// TwinCAT 3 PLC project WF03
// ProgramVersion: 3.1.4024.0
// libraries:
//   Tc2_Standard, * (Beckhoff Automation GmbH)
//   Tc2_System, * (Beckhoff Automation GmbH)
//   Tc3_Module, * (Beckhoff Automation GmbH)
// project tree:
//   DUTs/ E_ServoStateMachine.TcDUT, E_State.TcTLEO, E_ComponentMode.TcTLEO (not stored), E_LenzeJogFreq.TcTLEO, E_RotationDirection.TcTLEO (not stored)
//   GVLs/ GVL.TcGVL
//   / PlcTask.TcTTO (not stored), RevolutionCounter.TcTTO
//   POUs/deprecated/ FB_Module_4posArm_Old.TcPOU (not stored), FB_Module_CoilHolder_Old.TcPOU, FB_Module_ToolHolderDoor_Old.TcPOU, FB_Module_ToolHolder_Old.TcPOU
//   POUs/FB_Components/ FB_Component_ACmotor.TcPOU, FB_Component_DualValve.TcPOU, FB_Component_DualValveGuarded.TcPOU, FB_Component_InductiveSensor.TcPOU, FB_Component_ReedSwitch.TcPOU, FB_Component_Servo.TcPOU, FB_Component_SingleValve.TcPOU, FB_Component_SingleValveGuarded.TcPOU, FB_Component_4posArm.TcPOU
//   POUs/ COUNTER.TcPOU, FB_Component_ServoMotor.TcPOU, FB_Module_CoilPusher.TcPOU, FB_Section_Cutter.TcPOU, FB_Section_ToolStation_Old.TcPOU, I_Component.TcIO, I_Module.TcIO, I_Section.TcIO, MAIN.TcPOU
//   POUs/FB_Modules/ FB_Module_CoilHolder.TcPOU, FB_Module_ToolHolder.TcPOU, FB_Module_ToolHolderDoor.TcPOU, FB_Module_Winder.TcPOU
// real-time tasks:
//   TASK PlcTask: cycle T#10ms, priority 20, ADS port 350
//   TASK RevolutionCounter: cycle T#2ms, priority 1, ADS port 351
// I/O:
//   DEVICE Device 1 (EtherCAT), AmsNetId 5.155.196.195.2.1
//     Term 1 (EK1200) [EK1200-5000 EtherCAT Power supply (2A E-Bus)]
//       Term 2 (EL1809) [EL1809 16Ch. Dig. Input 24V, 3ms]
//       Term 3 (EL1809) [EL1809 16Ch. Dig. Input 24V, 3ms]
//       Term 4 (EL1809) [EL1809 16Ch. Dig. Input 24V, 3ms]
//       Term 5 (EL1809) [EL1809 16Ch. Dig. Input 24V, 3ms]
//       Term 6 (EL2809) [EL2809 16Ch. Dig. Output 24V, 0.5A]
//       Term 7 (EL2809) [EL2809 16Ch. Dig. Output 24V, 0.5A]
//       Term 8 (EL2809) [EL2809 16Ch. Dig. Output 24V, 0.5A]
//       Term 20 (EL4032) [EL4032 2Ch. Ana. Output +/-10V, 12bit]
//       Term 21 (EL5112) [EL5112 2Ch. Inc. Encoder 5V (2xAB or 1xABC RS422,TTL)]
//       Term 21 (EL9011) [EL9011 End Terminal]
// variable links:
//   WF03/WF03 Instance <-> Device 1 (EtherCAT)/Term 1 (EK1200)/Term 2 (EL1809)
//     PlcTask Inputs/GVL.bDoorToolHolderDown <-> Channel 4/Input
//     PlcTask Inputs/GVL.bDoorToolHolderLock <-> Channel 3/Input
//     PlcTask Inputs/GVL.bWireClampRetracted <-> Channel 12/Input
//     PlcTask Inputs/GVL.bWireClampTransverse1Extended <-> Channel 14/Input
//     PlcTask Inputs/GVL.bWireClampTransverse2Extended <-> Channel 16/Input
//     PlcTask Inputs/GVL.bWireClampTransverse1Retracted <-> Channel 13/Input
//     PlcTask Inputs/GVL.bWireClampTransverse2Retracted <-> Channel 15/Input
//     PlcTask Inputs/GVL.bWirePusherDisengaged <-> Channel 1/Input
//     PlcTask Inputs/GVL.bWirePusherEngaged <-> Channel 2/Input
//   WF03/WF03 Instance <-> Device 1 (EtherCAT)/Term 1 (EK1200)/Term 20 (EL4032)
//     PlcTask Outputs/GVL.aOutServo1 <-> AO Outputs Channel 1/Analog output
//     PlcTask Outputs/GVL.aOutServo2 <-> AO Outputs Channel 2/Analog output
//   WF03/WF03 Instance <-> Device 1 (EtherCAT)/Term 1 (EK1200)/Term 21 (EL5112)
//     PlcTask Inputs/GVL.bSetCounterDoneServo1 <-> ENC Status Channel 2/Status/Set counter done
//     PlcTask Inputs/GVL.bSetCounterDoneServo2 <-> ENC Status Channel 1/Status/Set counter done
//     PlcTask Inputs/GVL.dCountServo1 <-> ENC Status Channel 2/Counter value
//     PlcTask Outputs/GVL.dSetCounterServo1 <-> ENC Control Channel 2/Control/Set counter
//     PlcTask Outputs/GVL.dSetCounterServo2 <-> ENC Control Channel 1/Control/Set counter
//     PlcTask Outputs/GVL.dSetCounterValueServo1 <-> ENC Control Channel 2/Set counter value
//     PlcTask Outputs/GVL.dSetCounterValueServo2 <-> ENC Control Channel 1/Set counter value
//     RevolutionCounter Inputs/GVL.dCountServo2 <-> ENC Status Channel 1/Counter value
//   WF03/WF03 Instance <-> Device 1 (EtherCAT)/Term 1 (EK1200)/Term 3 (EL1809)
//     PlcTask Inputs/GVL.bCoilHolderIndexBit{1..5} <-> Channel {1..5}/Input  (5 links)
//     PlcTask Inputs/GVL.bCoilHolderIndexReady <-> Channel 6/Input
//     PlcTask Inputs/GVL.bCoilHolderLocked <-> Channel 8/Input
//     PlcTask Inputs/GVL.bCoilHolderUnlocked <-> Channel 7/Input
//     PlcTask Inputs/GVL.bToolHolderIndexBit1 <-> Channel 9/Input
//     PlcTask Inputs/GVL.bToolHolderIndexBit2 <-> Channel 10/Input
//     PlcTask Inputs/GVL.bToolHolderLocked <-> Channel 12/Input
//     PlcTask Inputs/GVL.bToolHolderUnlocked <-> Channel 11/Input
//     PlcTask Inputs/GVL.bWireHolderPos{1..4} <-> Channel {13..16}/Input  (4 links)
//   WF03/WF03 Instance <-> Device 1 (EtherCAT)/Term 1 (EK1200)/Term 4 (EL1809)
//     PlcTask Inputs/GVL.bCoilPusherExtended <-> Channel 2/Input
//     PlcTask Inputs/GVL.bCoilPusherRetracted <-> Channel 1/Input
//     PlcTask Inputs/GVL.bMainPressureSense <-> Channel 16/Input
//     PlcTask Inputs/GVL.bWire{1..4}NotAvailable <-> Channel {5..8}/Input  (4 links)
//   WF03/WF03 Instance <-> Device 1 (EtherCAT)/Term 1 (EK1200)/Term 5 (EL1809)
//     PlcTask Inputs/GVL.bCoilTranslate <-> Channel 15/Input
//     PlcTask Inputs/GVL.bControlOnBtn <-> Channel 5/Input
//     PlcTask Inputs/GVL.bFeedBackSafetyRelay <-> Channel 6/Input
//     PlcTask Inputs/GVL.bLenze1Relay <-> Channel 13/Input
//     PlcTask Inputs/GVL.bLenze2Relay <-> Channel 14/Input
//     PlcTask Inputs/GVL.bReadyToOperate603 <-> Channel 11/Input
//     PlcTask Inputs/GVL.bReadyToOperate614 <-> Channel 12/Input
//     PlcTask Inputs/GVL.bSafetyContactBreakers <-> Channel 9/Input
//     PlcTask Inputs/GVL.bStartBtn <-> Channel 2/Input
//     PlcTask Inputs/GVL.bStartPosBtn <-> Channel 3/Input
//     PlcTask Inputs/GVL.bStopBtn <-> Channel 1/Input
//     PlcTask Inputs/GVL.bToolingRotationBtn <-> Channel 4/Input
//     RevolutionCounter Inputs/GVL.bCoilRotate <-> Channel 16/Input
//   WF03/WF03 Instance <-> Device 1 (EtherCAT)/Term 1 (EK1200)/Term 6 (EL2809)
//     PlcTask Outputs/GVL.b603Enable <-> Channel 9/Output
//     PlcTask Outputs/GVL.b614Enable <-> Channel 10/Output
//     PlcTask Outputs/GVL.bCloseToolCarrierDoor <-> Channel 15/Output
//     PlcTask Outputs/GVL.bLenze1Direction <-> Channel 4/Output
//     PlcTask Outputs/GVL.bLenze1InjectionBrake <-> Channel 3/Output
//     PlcTask Outputs/GVL.bLenze1JogBit1 <-> Channel 1/Output
//     PlcTask Outputs/GVL.bLenze1JogBit2 <-> Channel 2/Output
//     PlcTask Outputs/GVL.bLenze2JogBit1 <-> Channel 5/Output
//     PlcTask Outputs/GVL.bLenze2JogBit2 <-> Channel 6/Output
//     PlcTask Outputs/GVL.bLenze2njectionBrake <-> Channel 7/Output
//     PlcTask Outputs/GVL.bOpenToolCarrierDoor <-> Channel 14/Output
//     PlcTask Outputs/GVL.bPushCoil <-> Channel 16/Output
//     PlcTask Outputs/GVL.bResetServosErrors <-> Channel 8/Output
//     PlcTask Outputs/GVL.bStartBtnLight <-> Channel 11/Output
//     PlcTask Outputs/GVL.bStartPosBtnLight <-> Channel 12/Output
//     PlcTask Outputs/GVL.bToolingRotationBtnLight <-> Channel 13/Output
//   WF03/WF03 Instance <-> Device 1 (EtherCAT)/Term 1 (EK1200)/Term 7 (EL2809)
//     PlcTask Outputs/GVL.bEngageWireClamp <-> Channel 12/Output
//     PlcTask Outputs/GVL.bExtendWireClamp <-> Channel 7/Output
//     PlcTask Outputs/GVL.bExtendWireHolder <-> Channel 5/Output
//     PlcTask Outputs/GVL.bExtendWireHolderTransverse1 <-> Channel 16/Output
//     PlcTask Outputs/GVL.bExtendWireHolderTransverse2 <-> Channel 9/Output
//     PlcTask Outputs/GVL.bLockDoor <-> Channel 2/Output
//     PlcTask Outputs/GVL.bReleaseWireClamp <-> Channel 11/Output
//     PlcTask Outputs/GVL.bRetractWireClamp <-> Channel 6/Output
//     PlcTask Outputs/GVL.bRetractWireHolder <-> Channel 4/Output
//     PlcTask Outputs/GVL.bRetractWireHolderTransverse1 <-> Channel 15/Output
//     PlcTask Outputs/GVL.bRetractWireHolderTransverse2 <-> Channel 8/Output
//     PlcTask Outputs/GVL.bUnlockCoilHolder <-> Channel 13/Output
//     PlcTask Outputs/GVL.bUnlockToolHolder <-> Channel 14/Output
//     PlcTask Outputs/GVL.bWirePusherForward <-> Channel 10/Output
//   WF03/WF03 Instance <-> Device 1 (EtherCAT)/Term 1 (EK1200)/Term 8 (EL2809)
//     PlcTask Outputs/GVL.bCutWire <-> Channel 1/Output

CONFIGURATION WF03
    RESOURCE PLC ON TwinCAT3
        TASK RevolutionCounter(INTERVAL := T#2ms, PRIORITY := 1);
        PROGRAM COUNTER WITH RevolutionCounter : COUNTER;
    END_RESOURCE
END_CONFIGURATION

// ---- DUTs/E_ServoStateMachine.TcDUT
{attribute 'qualified_only'}
{attribute 'strict'}
TYPE E_ServoStateMachine :
(
	IDLE			:= 0,
	HOMING          := 1,
	HOMED           := 2,
	RAMPUP          := 3,
	HOLD            := 4,
	RAMPDOWN        := 5,
	FAULT			:= 6
);
END_TYPE

// ---- DUTs/E_State.TcTLEO
{attribute 'qualified_only'}
{attribute 'strict'}
TYPE E_State :
(
	DISABLED	:= 0,
	READY		:= 1,
	BUSY		:= 2,
	DONE 		:= 3,
	HALTED		:= 4,
	TIMEOUT 	:= 5
);
END_TYPE

// ---- DUTs/E_LenzeJogFreq.TcTLEO
{attribute 'qualified_only'}
{attribute 'strict'}
TYPE E_LenzeJogFreq :
(
	FOFF 	:= 0,
	F1		:= 1,
	F2		:= 2,
	F3		:= 3
);
END_TYPE

// ---- GVLs/GVL.TcGVL
{attribute 'qualified_only'}
VAR_GLOBAL
	uRevCount1		: INT;
	uRevCount2		: DINT;
	bResetRevCount	: BOOL;

/////////////////////////////////////////////////////////////////////////////////////////////
// 									DIGITAL INPUTS								   		   //
/////////////////////////////////////////////////////////////////////////////////////////////
	//--------------------------------
	// TERM 2 : EL1809 Digital In
	//--------------------------------
	bWirePusherDisengaged			AT %I*	: BOOL;	// S5.18	term 2.1
	bWirePusherEngaged				AT %I*	: BOOL;	// S5.17	term 2.2
	bDoorToolHolderLock				AT %I*	: BOOL;	//			term 2.3
	bDoorToolHolderDown				AT %I*	: BOOL;	// S5.20	term 2.4
	// term 2.5-11 --> unused
	bWireClampRetracted				AT %I*	: BOOL;	// S5.28	term 2.12
	bWireClampTransverse1Extended	AT %I*	: BOOL;	// S5.29	term 2.14
	bWireClampTransverse1Retracted	AT %I*	: BOOL;	// S5.30	term 2.13
	bWireClampTransverse2Extended	AT %I*	: BOOL;	// S5.31	term 2.16
	bWireClampTransverse2Retracted	AT %I*	: BOOL;	// S5.32	term 2.15
	//--------------------------------
	// TERM 3 : EL1809 Digital In
	//--------------------------------
	bCoilHolderIndexBit1			AT %I*	: BOOL;	// S5.1		term 3.1
	bCoilHolderIndexBit2			AT %I*	: BOOL;	// S5.2		term 3.2
	bCoilHolderIndexBit3			AT %I*	: BOOL;	// S5.3		term 3.3
	bCoilHolderIndexBit4			AT %I*	: BOOL;	// S5.4		term 3.4
	bCoilHolderIndexBit5			AT %I*	: BOOL;	// S5.5		term 3.5
	bCoilHolderIndexReady			AT %I*	: BOOL;	// S5.6		term 3.6
	bCoilHolderUnlocked				AT %I*	: BOOL; // S5.8		term 3.7	
	bCoilHolderLocked				AT %I*	: BOOL; // S5.7		term 3.8
	bToolHolderIndexBit1			AT %I*	: BOOL; // S5.9		term 3.9
	bToolHolderIndexBit2			AT %I*	: BOOL; // S5.10	term 3.10
	bToolHolderUnlocked				AT %I*	: BOOL; // S5.12	term 3.11
	bToolHolderLocked   			AT %I*	: BOOL; // S5.11	term 3.12
	bWireHolderPos1					AT %I*	: BOOL; // S5.13	term 3.13
	bWireHolderPos2					AT %I*	: BOOL; // S5.14	term 3.14
	bWireHolderPos3					AT %I*	: BOOL; // S5.15	term 3.15
	bWireHolderPos4					AT %I*	: BOOL; // S5.16	term 3.16
	//--------------------------------
	// TERM 4 : EL1809 Digital In
	//--------------------------------
	bCoilPusherRetracted			AT %I*	: BOOL;	// S4.17	term 4.1
	bCoilPusherExtended				AT %I*	: BOOL;	// S4.18	term 4.2
	// term 4.3-4 --> unused
	bWire1NotAvailable				AT %I*	: BOOL;	// S4.21	term 4.5
	bWire2NotAvailable				AT %I*	: BOOL;	// S4.22	term 4.6
	bWire3NotAvailable				AT %I*	: BOOL;	// S4.23	term 4.7
	bWire4NotAvailable				AT %I*	: BOOL;	// S4.24	term 4.8
	// term 4.9-15 --> unused
	bMainPressureSense				AT %I*	: BOOL;	// S4.32	term 4.16
	//--------------------------------
	// TERM 5 : EL1809 Digital In
	//--------------------------------
	bStopBtn						AT %I*	: BOOL;	//			term 5.1
	bStartBtn						AT %I*	: BOOL;	//			term 5.2
	bStartPosBtn					AT %I*	: BOOL;	//			term 5.3
	bToolingRotationBtn				AT %I*	: BOOL;	//			term 5.4
	bControlOnBtn					AT %I*	: BOOL;	//			term 5.5
	bFeedBackSafetyRelay			AT %I*	: BOOL; //			term 5.6
	// term 5.7 check why connected to GND											// TODO!!
	// term 5.8	check what contactor K1.1 does and if also checks other stuff		// TODO!!
	bSafetyContactBreakers			AT %I*	: BOOL;	//			term 5.9
	// term 5.10 --> unused
	bReadyToOperate603				AT %I*	: BOOL;	//			term 5.11			// rename
	bReadyToOperate614				AT %I*	: BOOL;	//			term 5.12			// rename
	bLenze1Relay					AT %I*	: BOOL;	//			term 5.13			// rename
	bLenze2Relay					AT %I*	: BOOL;	//			term 5.14			// rename
	bCoilTranslate					AT %I*	: BOOL;	//			term 5.15			// rename
	bCoilRotate						AT %I*	: BOOL;	//			term 5.16			// rename

/////////////////////////////////////////////////////////////////////////////////////////////
// 									DIGITAL OUTPUTS								   		   //
/////////////////////////////////////////////////////////////////////////////////////////////
	//--------------------------------
	// TERM 6 : EL2809 Digital Out
	//--------------------------------
	bLenze1JogBit1					AT %Q*	: BOOL;	//			term 6.1
	bLenze1JogBit2					AT %Q*	: BOOL;	//			term 6.2
	bLenze1InjectionBrake			AT %Q*	: BOOL; //			term 6.3
	bLenze1Direction				AT %Q*	: BOOL;	//			term 6.4
	bLenze2JogBit1					AT %Q*	: BOOL;	//			term 6.5
	bLenze2JogBit2					AT %Q*	: BOOL;	//			term 6.6
	bLenze2njectionBrake			AT %Q*	: BOOL; //			term 6.7
	bResetServosErrors				AT %Q*	: BOOL; //			term 6.8
	b603Enable						AT %Q*	: BOOL;	//			term 6.9
	b614Enable						AT %Q*	: BOOL;	//			term 6.10
	bStartBtnLight					AT %Q*	: BOOL; //			term 6.11
	bStartPosBtnLight				AT %Q*	: BOOL; //			term 6.12
	bToolingRotationBtnLight		AT %Q*	: BOOL; //			term 6.13
	bOpenToolCarrierDoor			AT %Q*	: BOOL; // Y6.4		term 6.14
	bCloseToolCarrierDoor			AT %Q*	: BOOL; // Y6.5		term 6.15
	bPushCoil						AT %Q*	: BOOL; // Y6.9		term 6.16
	//--------------------------------
	// TERM 7 : EL2809 Digital Out
	//--------------------------------
	// term 7.1 --> unused
	bLockDoor						AT %Q*	: BOOL; //			term 7.2
	// term 7.3 --> unused
	bRetractWireHolder				AT %Q*	: BOOL; // Y6.13	term 7.4
	bExtendWireHolder				AT %Q*	: BOOL; // Y6.14	term 7.5
	bRetractWireClamp				AT %Q*	: BOOL; // Y7.10	term 7.6		// pushes forward clamp
	bExtendWireClamp				AT %Q*	: BOOL; // Y7.11	term 7.7
	bRetractWireHolderTransverse2	AT %Q*	: BOOL; // Y7.7		term 7.8
	bExtendWireHolderTransverse2	AT %Q*	: BOOL; // Y7.8		term 7.9
	bWirePusherForward				AT %Q*	: BOOL; // Y7.9		term 7.10		// bent thingy pushing the wire at the top
	bReleaseWireClamp				AT %Q*	: BOOL; // Y6.15	term 7.11		// clamps wire
	bEngageWireClamp				AT %Q*	: BOOL; // Y6.16	term 7.12
	bUnlockCoilHolder				AT %Q*	: BOOL; // Y7.12	term 7.13
	bUnlockToolHolder				AT %Q*	: BOOL; // Y7.13	term 7.14
	bRetractWireHolderTransverse1	AT %Q*	: BOOL; // Y7.14	term 7.15
	bExtendWireHolderTransverse1	AT %Q*	: BOOL; // Y7.15	term 7.16
	//--------------------------------
	// TERM 8 : EL2809 Digital Out
	//--------------------------------
	bCutWire						AT %Q*	: BOOL; // Y8.1		term 7.1
	// term 8.2-9 --> unused
	// term 8.16-16 --> free
	
	//--------------------------------
	// TERM 8 : EL4032 Analog Out
	//--------------------------------
	aOutServo1						AT %Q*	: INT;	// term 20
	aOutServo2						AT %Q*	: INT;	// term 20
	
	bSetCounterDoneServo1			AT %I*	: BOOL;	// term 21
	dCountServo1					AT %I*	: DINT;	// term 21
	bSetCounterDoneServo2			AT %I*	: BOOL;	// term 21
	dCountServo2					AT %I*	: DINT;	// term 21
	
	dSetCounterServo1				AT %Q*	: BOOL;	// term 21
	dSetCounterValueServo1			AT %Q*	: DINT;	// term 21
	dSetCounterServo2				AT %Q*	: BOOL;	// term 21
	dSetCounterValueServo2			AT %Q*	: DINT;	// term 21
	
END_VAR

// ---- POUs/I_Component.TcIO
INTERFACE I_Component
VAR_INPUT
END_VAR

VAR_OUTPUT
END_VAR

METHOD M_Disable : BOOL
VAR_INPUT
END_VAR
END_METHOD

METHOD M_Enable : BOOL
VAR_INPUT
END_VAR
END_METHOD

METHOD M_Halt : BOOL
VAR_INPUT
END_VAR
END_METHOD

METHOD M_Resume : BOOL
VAR_INPUT
END_VAR
END_METHOD

END_INTERFACE

// ---- POUs/I_Module.TcIO
INTERFACE I_Module

METHOD M_Disable : BOOL
VAR_INPUT
END_VAR
END_METHOD

METHOD M_Enable : BOOL
VAR_INPUT
END_VAR
END_METHOD

METHOD M_Halt : BOOL
VAR_INPUT
END_VAR
END_METHOD

METHOD M_Resume : BOOL
VAR_INPUT
END_VAR
END_METHOD

END_INTERFACE

// ---- POUs/I_Section.TcIO
INTERFACE I_Section

METHOD M_Disable : BOOL
VAR_INPUT
END_VAR
END_METHOD

METHOD M_Enable : BOOL
VAR_INPUT
END_VAR
END_METHOD

METHOD M_Halt : BOOL
VAR_INPUT
END_VAR
END_METHOD

METHOD M_Resume : BOOL
VAR_INPUT
END_VAR
END_METHOD

END_INTERFACE

// ---- POUs/COUNTER.TcPOU
PROGRAM COUNTER
VAR
	tSensorTrig		: F_TRIG;
END_VAR

tSensorTrig(CLK := GVL.bCoilRotate);
IF tSensorTrig.Q THEN
	GVL.uRevCount1 := GVL.uRevCount1 + 1;
END_IF

IF GVL.bResetRevCount THEN
	GVL.bResetRevCount  := FALSE;
	GVL.uRevCount1		:= 0;
END_IF

GVL.uRevCount2 := REAL_TO_DINT(DINT_TO_REAL(GVL.dCountServo2) / 9216);

END_PROGRAM

// ---- POUs/deprecated/FB_Module_CoilHolder_Old.TcPOU
FUNCTION_BLOCK FB_Module_CoilHolder_Old IMPLEMENTS I_Module
VAR_INPUT
	bEnable			: BOOL;
END_VAR
VAR_OUTPUT
END_VAR
VAR
	Components		: ARRAY [0..9] OF I_Component;

	fbACmotor		: FB_Component_ACmotor;
	fbCoilLock		: FB_Component_SingleValve;
	fbReedLock		: FB_Component_ReedSwitch;
	fbReedUnlock	: FB_Component_ReedSwitch;
	
	fbIndexBit1		: FB_Component_InductiveSensor;
	fbIndexBit2		: FB_Component_InductiveSensor;
	fbIndexBit3		: FB_Component_InductiveSensor;
	fbIndexBit4		: FB_Component_InductiveSensor;
	fbIndexBit5		: FB_Component_InductiveSensor;
	fbIndexReady	: FB_Component_InductiveSensor;
	
	nIndex			: INT;
	idx				: INT;
END_VAR

IF bEnable THEN
	fbACmotor(
		bDeviceActive 	:= GVL.bLenze1Relay,
		sName			:= 'AC motor plate',
		bEnable			:= TRUE,
		bE1jog1			:= GVL.bLenze1JogBit1,
		bE2jog2			:= GVL.bLenze1JogBit2,
		bE3DCbrake		:= GVL.bLenze1InjectionBrake,
		eE4Direction	:= GVL.bLenze1Direction);
		
	fbCoilLock(
		sName 	:= 'Coil Lock',
		bEnable := TRUE,
		bOutput := GVL.bUnlockCoilHolder);
		
	fbReedLock(
		bRawSignal	:= GVL.bCoilHolderLocked,
		tDebounce	:= T#5MS,
		tTimeout	:= T#0S,
		sName		:= 'plate locked reed',
		bEnable		:= TRUE);
		
	fbReedUnlock(
		bRawSignal	:= GVL.bCoilHolderUnlocked,
		tDebounce	:= T#5MS,
		tTimeout	:= T#0S,
		sName		:= 'plate unlocked reed',
		bEnable		:= TRUE);
		
	fbIndexBit1(bRawSignal := GVL.bCoilHolderIndexBit1,
		tDebounce 	:= T#5MS,
		tTimeout	:= T#0S,
		sName		:= 'plate index 1',
		bEnable		:= TRUE);
		
	fbIndexBit2(bRawSignal := GVL.bCoilHolderIndexBit2,
		tDebounce 	:= T#5MS,
		tTimeout	:= T#0S,
		sName		:= 'plate index 2',
		bEnable		:= TRUE);
		
	fbIndexBit3(bRawSignal := GVL.bCoilHolderIndexBit3,
		tDebounce 	:= T#5MS,
		tTimeout	:= T#0S,
		sName		:= 'plate index 3',
		bEnable		:= TRUE);
		
	fbIndexBit4(bRawSignal := GVL.bCoilHolderIndexBit4,
		tDebounce 	:= T#5MS,
		tTimeout	:= T#0S,
		sName		:= 'plate index 4',
		bEnable		:= TRUE);
		
	fbIndexBit5(bRawSignal := GVL.bCoilHolderIndexBit5,
		tDebounce 	:= T#5MS,
		tTimeout	:= T#0S,
		sName		:= 'plate index 5',
		bEnable		:= TRUE);
		
	fbIndexReady(bRawSignal := GVL.bCoilHolderIndexReady,
		tDebounce 	:= T#5MS,
		tTimeout	:= T#0S,
		sName		:= 'plate index ready',
		bEnable		:= TRUE);

	Components[0] := fbACmotor;
	Components[1] := fbCoilLock;
	Components[2] := fbReedLock;
	Components[3] := fbReedUnlock;
	Components[4] := fbIndexBit1;
	Components[5] := fbIndexBit2;
	Components[6] := fbIndexBit3;
	Components[7] := fbIndexBit4;
	Components[8] := fbIndexBit5;
	Components[9] := fbIndexReady;
	
	FOR idx := 0 TO 9 DO
    	Components[idx].M_Start();
	END_FOR;
	
	// when index ready bit is triggered, convert index bits to integer
	IF fbIndexReady.bSensorActive THEN
		nIndex := 	TO_INT(SHL(TO_UINT(fbIndexBit5.bSensorActive), 4) OR
					SHL(TO_UINT(fbIndexBit4.bSensorActive), 3) OR
					SHL(TO_UINT(fbIndexBit3.bSensorActive), 2) OR
					SHL(TO_UINT(fbIndexBit2.bSensorActive), 1) OR
					(TO_UINT(fbIndexBit1.bSensorActive)));
	END_IF
END_IF

METHOD M_GoTo : BOOL
VAR_INPUT
	nTargetIndex	: INT;
END_VAR

VAR
	cwSteps: INT;
	target: INT;
	ccwSteps: INT;
	shortestDistance : INT;
END_VAR
IF fbReedUnlock.bSensorActive THEN
	IF nTargetIndex = nIndex THEN									// if target index is reached, turn off motor, lock plate and signal done
		fbACmotor.M_SetFreq(Frequency := E_LenzeJogFreq.F0FF);
		M_Lock();
		M_GoTo := TRUE;
		RETURN;
	END_IF
	
	cwSteps  := (nTargetIndex - nIndex + 24) MOD 24;				// calculate how much cw & ccw steps needed to go to target
	ccwSteps := (nIndex - nTargetIndex + 24) MOD 24;
	
	IF cwSteps <= ccwSteps THEN										// set direction for shortest path to target
		fbACmotor.M_SetDir(Direction := E_RotationDirection.CW);
		shortestDistance := cwSteps;
	ELSE
		fbACmotor.M_SetDir(Direction := E_RotationDirection.CCW);	
		shortestDistance := ccwSteps;
	END_IF
	
	IF nIndex <> nTargetIndex THEN
		IF shortestDistance <= 1 THEN								// if 1 from the target, set speed to slowest
			fbACmotor.M_SetFreq(Frequency := E_LenzeJogFreq.F1);	
		ELSIF shortestDistance <= 2 THEN							// if 2 from the target, set speed to slow
			fbACmotor.M_SetFreq(Frequency := E_LenzeJogFreq.F2);
		ELSE
			fbACmotor.M_SetFreq(Frequency := E_LenzeJogFreq.F3);	// if further set to highest speed
		END_IF
	ELSE
		fbACmotor.M_SetFreq(Frequency := E_LenzeJogFreq.F0FF);		// for safety, should be handled by first if
		M_Lock();
		M_GoTo := TRUE;
	END_IF
ELSE
	M_Unlock();														// unlock plate if locked
END_IF
END_METHOD

METHOD M_Halt : BOOL
VAR_INPUT
END_VAR
END_METHOD

METHOD M_Lock : BOOL
VAR_INPUT
END_VAR
fbCoilLock.M_Retract();
END_METHOD

METHOD M_Start : BOOL
VAR_INPUT
END_VAR
END_METHOD

METHOD M_Stop : BOOL
VAR_INPUT
END_VAR
END_METHOD

METHOD M_Unlock : BOOL
VAR_INPUT
END_VAR
fbCoilLock.M_Extend();
END_METHOD

END_FUNCTION_BLOCK

// ---- POUs/FB_Components/FB_Component_ACmotor.TcPOU
// Function block for AC motors controlled with the LENZE d-31855 frequency inverter
FUNCTION_BLOCK FB_Component_ACmotor IMPLEMENTS I_Component
VAR_INPUT
	sName			: STRING[50];
	tTimeout		: TIME := T#0MS;
END_VAR

VAR_OUTPUT
	eJogFreq		: E_LenzeJogFreq := E_LenzeJogFreq.FOFF;
	
	bEnabled     	: BOOL;
	eState			: E_State := E_State.DISABLED;
	eNextState		: E_State := E_State.DISABLED;
	sStatusText 	: STRING[100];
END_VAR

VAR_IN_OUT
	bDeviceActive	: BOOL;	
	bE1jog1			: BOOL;					// jog func b1
	bE2jog2			: BOOL;					// jog func b2
	bE3DCbrake		: BOOL;					// DC injection brake
	eE4Direction	: BOOL;					// motor direction
END_VAR

VAR
	bLastE1jog1		: BOOL;
	bLastE2jog2		: BOOL;
	eLastState		: E_State;
	tTimeoutTimer	: TON;
END_VAR


VAR CONSTANT
	DISABLED		: E_State := E_State.DISABLED;
	READY			: E_State := E_State.READY;
	BUSY			: E_State := E_State.BUSY;
	HALTED			: E_State := E_State.HALTED;
	TIMEOUT			: E_State := E_State.TIMEOUT;
	
	FOFF	: E_LenzeJogFreq := E_LenzeJogFreq.FOFF;
	F1		: E_LenzeJogFreq := E_LenzeJogFreq.F1;
	F2		: E_LenzeJogFreq := E_LenzeJogFreq.F2;
	F3		: E_LenzeJogFreq := E_LenzeJogFreq.F3;
END_VAR

tTimeoutTimer(PT := tTimeout);

eState := eNextState;

CASE eState OF
	DISABLED:	sStatusText := 'AC motor disabled';
	
	READY:	 	sStatusText := 'Motor not moving, waiting for instruction';
				IF NOT bDeviceActive THEN
					sStatusText := 'frequency inverter is not activated, please check if control is on and doors are closed';
				ELSIF eJogFreq <> FOFF THEN
					eNextState := BUSY;
				END_IF
				
	BUSY: 		M_ApplyFreq();
				CASE eJogFreq OF
					FOFF: 	eNextState	:= E_State.TIMEOUT;
					F1: 	sStatusText := CONCAT('motor running ', CONCAT(SEL(eE4Direction = TRUE, 'CCW','CW'), ' at freq 1'));		
					F2: 	sStatusText := CONCAT('motor running ', CONCAT(SEL(eE4Direction = TRUE, 'CCW','CW'), ' at freq 2'));				
					F3: 	sStatusText := CONCAT('motor running ', CONCAT(SEL(eE4Direction = TRUE, 'CCW','CW'), ' at freq 3')); 	
				END_CASE
	
	TIMEOUT: 	sStatusText := 'motor in timeout';
				tTimeoutTimer(IN := TRUE);
				
				IF tTimeoutTimer.Q THEN
					tTimeoutTimer(IN := FALSE);
					eNextState := READY;
				END_IF
	
	HALTED: 	sStatusText := 'motor halted';

END_CASE

METHOD M_ApplyFreq : BOOL
VAR_INPUT
END_VAR
IF eState = BUSY AND bDeviceActive THEN
	CASE eJogFreq OF
		FOFF: 	bE1jog1 	:= FALSE;
				bE2jog2 	:= FALSE;
				
		F1: 	bE1jog1 	:= TRUE;
				bE2jog2 	:= FALSE;
				
		F2: 	bE1jog1 	:= TRUE;
				bE2jog2 	:= TRUE;

		F3: 	bE1jog1 	:= FALSE;
				bE2jog2 	:= TRUE;
	END_CASE
END_IF
END_METHOD

METHOD M_Disable : BOOL
VAR_INPUT
END_VAR
IF eState = READY THEN
	bE1jog1		 	:= FALSE;
	bE2jog2		 	:= FALSE;
	bE3DCbrake 		:= FALSE;
	eE4Direction 	:= FALSE;
	tTimeoutTimer(IN := FALSE);	

	bEnabled	:= FALSE;
	eNextState	:= DISABLED;
END_IF
END_METHOD

METHOD M_Enable : BOOL
VAR_INPUT
END_VAR
IF eState = DISABLED THEN
	bEnabled	:= TRUE;
	eNextState 	:= READY;
END_IF
END_METHOD

METHOD M_Halt : BOOL
VAR_INPUT
END_VAR
IF eState <> HALTED AND eState <> DISABLED THEN
	bLastE1jog1 := bE1jog1;
	bLastE2jog2 := bE2jog2;
	
	bE1jog1		:= FALSE;
	bE2jog2		:= FALSE;
	bE3DCbrake	:= TRUE;
	
	eLastState 	:= eState;
	eNextState 	:= HALTED;	
END_IF
END_METHOD

METHOD M_Resume : BOOL
VAR_INPUT
END_VAR
IF eState = HALTED THEN
	bE1jog1 	:= bLastE1jog1;
	bE2jog2 	:= bLastE2jog2;
	bE3DCbrake 	:= FALSE;
	
	eNextState 	:= eLastState;
END_IF
END_METHOD

METHOD M_SetDir : BOOL
VAR_INPUT
	Direction: E_RotationDirection;
END_VAR
IF eState = READY THEN
	eE4Direction := TO_BOOL(Direction);
END_IF
END_METHOD

METHOD M_SetFreq : BOOL
VAR_INPUT
	Frequency: E_LenzeJogFreq;
END_VAR
IF eState = READY OR eState = BUSY THEN
	eJogFreq := Frequency;
END_IF
END_METHOD

END_FUNCTION_BLOCK

// ---- POUs/FB_Components/FB_Component_SingleValve.TcPOU
FUNCTION_BLOCK FB_Component_SingleValve IMPLEMENTS I_Component
VAR_INPUT
	sName			: STRING[50];
	tTimeout		: TIME := T#0S;
END_VAR

VAR_IN_OUT
	bOutput			: BOOL;
END_VAR

VAR_OUTPUT
	bEnabled     	: BOOL;
	eState			: E_State := E_State.DISABLED;
	eNextState		: E_State := E_State.DISABLED;
	sStatusText 	: STRING[100];
END_VAR

VAR
	tTimeoutTimer	: TON;
	eLastState		: E_State;
END_VAR

VAR CONSTANT
	DISABLED		: E_State := E_State.DISABLED;
	READY			: E_State := E_State.READY;
	BUSY			: E_State := E_State.BUSY;
	HALTED			: E_State := E_State.HALTED;
	TIMEOUT			: E_State := E_State.TIMEOUT;
END_VAR

tTimeoutTimer(PT := tTimeout);

eState := eNextState;

CASE eState OF
	DISABLED: 	sStatusText := 'piston is disabled';
	READY: 		sStatusText := 'piston ready to operate';
	BUSY: 		sStatusText := 'piston busy';
	TIMEOUT:	sStatusText := 'piston in timeout';
				tTimeoutTimer(IN := TRUE);
				
				IF tTimeoutTimer.Q THEN
					tTimeoutTimer(IN := FALSE);
					eNextState := READY;
				END_IF
				
	HALTED:		sStatusText := 'piston halted';
END_CASE

METHOD M_Disable : BOOL
VAR_INPUT
END_VAR
IF eState = READY THEN
	bEnabled	:= FALSE;
	eNextState	:= DISABLED;
END_IF
END_METHOD

METHOD M_Enable : BOOL
VAR_INPUT
END_VAR
IF eState = DISABLED THEN
	bEnabled	:= TRUE;
	eNextState	:= READY;
END_IF
END_METHOD

METHOD M_Extend : BOOL
VAR_INPUT
END_VAR
IF eState = READY OR eState = BUSY THEN
	bOutput := TRUE;
END_IF
END_METHOD

METHOD M_Halt : BOOL
VAR_INPUT
END_VAR
IF eState <> HALTED AND eState <> DISABLED THEN
	eLastState := eState;
	eNextState := HALTED;
END_IF
END_METHOD

METHOD M_Resume : BOOL
VAR_INPUT
END_VAR
IF eState = HALTED THEN
	eNextState := eLastState;
END_IF
END_METHOD

METHOD M_Retract : BOOL
VAR_INPUT
END_VAR
IF eState = READY OR eState = BUSY THEN
	bOutput	:= FALSE;
END_IF
END_METHOD

END_FUNCTION_BLOCK

// ---- POUs/FB_Components/FB_Component_ReedSwitch.TcPOU
// function block for reed switch with the option of debouncing + rising and falling edge detection.
FUNCTION_BLOCK FB_Component_ReedSwitch IMPLEMENTS I_Component
VAR_INPUT
	sName			: STRING[50];
	bRawSignal		: BOOL;				
	tDebounce		: TIME := T#0MS;
	tTimeout		: TIME := T#0MS;
END_VAR

VAR_OUTPUT
	bSensorActive	: BOOL;
	bTimeout		: BOOL;
	bRisingEdge		: BOOL;
	bFallingEdge	: BOOL;
	
	bEnabled		: BOOL;
	eState			: E_State := E_State.DISABLED;
	eNextState		: E_State := E_State.DISABLED;
	sStatusText 	: STRING[100];
END_VAR

VAR
	tDebounceTimer		: TON;
	tTimeoutTimer		: TON;
	
	bLastStableSignal	: BOOL := bRawSignal;
	bPendingSignal		: BOOL;
	
	eLastState			: E_State;
END_VAR

VAR CONSTANT
	DISABLED	: E_State := E_State.DISABLED;
	READY		: E_State := E_State.READY;
	BUSY		: E_State := E_State.BUSY;
	DONE		: E_State := E_State.DONE;
	HALTED		: E_State := E_State.HALTED;
	TIMEOUT		: E_State := E_State.TIMEOUT;
END_VAR

tDebounceTimer.PT 	:= tDebounce;
tTimeoutTimer.PT	:= tTimeout;

eState := eNextState;

CASE eState OF
	DISABLED:	sStatusText := 'Sensor disabled';
				
	READY:		sStatusText := 'Sensor idle, waiting for read';
				IF bRawSignal <> bLastStableSignal THEN
					bPendingSignal 	:= bRawSignal;
					eNextState 		:= BUSY;
				ELSE
					tTimeoutTimer(IN := FALSE);
					tDebounceTimer(IN := FALSE);
				END_IF
				
	BUSY:		sStatusText := 'Sensor is debouncing';
				tDebounceTimer(IN := TRUE);
				IF bRawSignal <> bPendingSignal THEN
					eNextState := READY;
				END_IF

				IF tDebounceTimer.Q THEN
					eNextState := TIMEOUT;
				END_IF
	TIMEOUT:	sStatusText := 'Sensor timeout';
				tTimeoutTimer(IN := TRUE);
				
				bRisingEdge  := NOT bLastStableSignal AND bPendingSignal;
				bFallingEdge := bLastStableSignal AND NOT bPendingSignal;
					
				bLastStableSignal := bPendingSignal;
				bSensorActive	  := bLastStableSignal;
				
				IF tTimeoutTimer.Q THEN
					tTimeoutTimer(IN 	:= FALSE);
					tDebounceTimer(IN 	:= FALSE);
					eNextState := READY;
				END_IF
				
	HALTED:		sStatusText := 'Sensor halted';
								
END_CASE

METHOD M_Disable : BOOL
VAR_INPUT
END_VAR
IF eState = READY THEN
	bEnabled	:= FALSE;
	eNextState	:= DISABLED;
END_IF
END_METHOD

METHOD M_Enable : BOOL
VAR_INPUT
END_VAR
IF eState = DISABLED THEN
	bEnabled	:= TRUE;
	eNextState	:= READY;
END_IF
END_METHOD

METHOD M_Halt : BOOL
VAR_INPUT
END_VAR
tDebounceTimer(IN := FALSE);
eLastState 	:= eState;
eNextState	:= HALTED;
END_METHOD

METHOD M_ResetEdge : BOOL
VAR_INPUT
END_VAR
bRisingEdge		:= FALSE;
bFallingEdge	:= FALSE;
END_METHOD

METHOD M_Resume : BOOL
VAR_INPUT
END_VAR
IF eState = HALTED THEN
	eNextState := eLastState;
END_IF
END_METHOD

END_FUNCTION_BLOCK

// ---- POUs/FB_Components/FB_Component_InductiveSensor.TcPOU
// function block for inductive sensor with the option of debouncing + rising and falling edge detection.
FUNCTION_BLOCK FB_Component_InductiveSensor IMPLEMENTS  I_Component
VAR_INPUT
	sName			: STRING[50];
	bRawSignal		: BOOL;				
	tDebounce		: TIME := T#0MS;
	tTimeout		: TIME := T#0MS;
END_VAR

VAR_OUTPUT
	bSensorActive	: BOOL;
	bTimeout		: BOOL;
	bRisingEdge		: BOOL;
	bFallingEdge	: BOOL;
	
	bEnabled		: BOOL;
	eState			: E_State := E_State.DISABLED;
	eNextState			: E_State := E_State.DISABLED;
	sStatusText 	: STRING[100];
END_VAR

VAR
	tDebounceTimer		: TON;
	tTimeoutTimer		: TON;
	
	bLastStableSignal	: BOOL := bRawSignal;
	bPendingSignal		: BOOL;
	
	eLastState			: E_State;
END_VAR

VAR CONSTANT
	DISABLED	: E_State := E_State.DISABLED;
	READY		: E_State := E_State.READY;
	BUSY		: E_State := E_State.BUSY;
	HALTED		: E_State := E_State.HALTED;
	TIMEOUT		: E_State := E_State.TIMEOUT;
END_VAR

tDebounceTimer.PT 	:= tDebounce;
tTimeoutTimer.PT	:= tTimeout;

eState := eNextState;

CASE eState OF
	DISABLED:	sStatusText := 'Sensor disabled';
				
	READY:		sStatusText := 'Sensor idle, waiting for read';
				IF bRawSignal <> bLastStableSignal THEN
					bPendingSignal 	:= bRawSignal;
					eNextState 		:= BUSY;
				ELSE
					tTimeoutTimer(IN := FALSE);
					tDebounceTimer(IN := FALSE);
				END_IF
				
	BUSY:		sStatusText := 'Sensor is debouncing';
				tDebounceTimer(IN := TRUE);
				IF bRawSignal <> bPendingSignal THEN
					eNextState := READY;
				END_IF

				IF tDebounceTimer.Q THEN
					eNextState := TIMEOUT;
				END_IF
	TIMEOUT:	sStatusText := 'Sensor timeout';
				tTimeoutTimer(IN := TRUE);
				
				bRisingEdge  := NOT bLastStableSignal AND bPendingSignal;
				bFallingEdge := bLastStableSignal AND NOT bPendingSignal;
					
				bLastStableSignal := bPendingSignal;
				bSensorActive	  := bLastStableSignal;
				
				IF tTimeoutTimer.Q THEN
					tTimeoutTimer(IN 	:= FALSE);
					tDebounceTimer(IN 	:= FALSE);
					eNextState := READY;
				END_IF
				
	HALTED:		sStatusText := 'Sensor halted';
								
END_CASE

METHOD M_Disable : BOOL
VAR_INPUT
END_VAR
IF eState = READY THEN
	bEnabled	:= FALSE;
	eNextState	:= DISABLED;
END_IF
END_METHOD

METHOD M_Enable : BOOL
VAR_INPUT
END_VAR
IF eState = DISABLED THEN
	bEnabled	:= TRUE;
	eNextState	:= READY;
END_IF
END_METHOD

METHOD M_Halt : BOOL
VAR_INPUT
END_VAR
tDebounceTimer(IN := FALSE);
eLastState 	:= eState;
eNextState	:= HALTED;
END_METHOD

METHOD M_ResetEdge : BOOL
VAR_INPUT
END_VAR
bRisingEdge		:= FALSE;
bFallingEdge	:= FALSE;
END_METHOD

METHOD M_Resume : BOOL
VAR_INPUT
END_VAR
IF eState = HALTED THEN
	eNextState := eLastState;
END_IF
END_METHOD

END_FUNCTION_BLOCK

// ---- POUs/deprecated/FB_Module_ToolHolderDoor_Old.TcPOU
FUNCTION_BLOCK FB_Module_ToolHolderDoor_Old IMPLEMENTS I_Module
VAR_INPUT
	bEnable					: BOOL;
END_VAR
VAR_OUTPUT
	bDoorUp				: BOOL;
END_VAR
VAR
	Components			: ARRAY [0..2] OF I_Component;
	
	fbPiston			: FB_Component_DualValve;
	fbDoorUp			: FB_Component_InductiveSensor;
	fbDoorDown			: FB_Component_ReedSwitch;
	idx					: INT;
END_VAR

IF bEnable THEN
	fbPiston(
		sName 		:= 'door piston',
		bEnable		:= TRUE,
		bOutputA	:= GVL.bCloseToolCarrierDoor,
		bOutputB	:= GVL.bOpenToolCarrierDoor);
	
	fbDoorUp(
		bRawSignal	:= GVL.bDoorToolHolderLock,
		tDebounce	:= T#0MS,
		tTimeout	:= T#0MS,
		sName		:= 'door up',
		bEnable		:= TRUE);
		
	fbDoorDown(
		bRawSignal	:= GVL.bDoorToolHolderDown,
		tDebounce	:= T#0MS,
		tTimeout	:= T#0MS,
		sName		:= 'door down',
		bEnable		:= TRUE);
		
	Components[0]	:= fbPiston;
	Components[1]	:= fbDoorUp;
	Components[2]	:= fbDoorDown;
	
	FOR idx := 0 TO 2 DO
    	Components[idx].M_Start();
	END_FOR;
	
	bDoorUp := fbDoorUp.bSensorActive;
END_IF

METHOD M_Down : BOOL
VAR_INPUT
END_VAR
IF bEnable THEN
	IF fbDoorDown.bSensorActive THEN
		fbPiston.M_Hold();
		M_Down := TRUE;
	ELSE
		fbPiston.M_Retract();
	END_IF
END_IF
END_METHOD

{warning 'add method implementation '}
METHOD M_Halt : BOOL
END_METHOD

{warning 'add method implementation '}
METHOD M_Start : BOOL
END_METHOD

{warning 'add method implementation '}
METHOD M_Stop : BOOL
END_METHOD

METHOD M_Up : BOOL
VAR_INPUT
END_VAR
IF bEnable THEN
	IF fbDoorUp.bSensorActive THEN
		fbPiston.M_Hold();
		M_Up := TRUE;
	ELSE
		fbPiston.M_Extend();
	END_IF
END_IF
END_METHOD

END_FUNCTION_BLOCK

// ---- POUs/FB_Components/FB_Component_DualValve.TcPOU
FUNCTION_BLOCK FB_Component_DualValve IMPLEMENTS I_Component
VAR_INPUT
	sName			: STRING[50];
	tTimeout		: TIME := T#0S;
END_VAR

VAR_IN_OUT
	bOutputA		: BOOL;
	bOutputB		: BOOL;
END_VAR

VAR_OUTPUT
	bEnabled     	: BOOL;
	eState			: E_State := E_State.DISABLED;
	eNextState		: E_State := E_State.DISABLED;
	sStatusText 	: STRING[100];
END_VAR

VAR
	bStartTimeout	: BOOL;
	tTimeoutTimer	: TON;
	bLastOutputA	: BOOL;
	bLastOutputB	: BOOL;
	eLastState		: E_State;
END_VAR

VAR CONSTANT
	DISABLED		: E_State := E_State.DISABLED;
	READY			: E_State := E_State.READY;
	BUSY			: E_State := E_State.BUSY;
	DONE			: E_State := E_State.DONE;
	HALTED			: E_State := E_State.HALTED;
	TIMEOUT			: E_State := E_State.TIMEOUT;
END_VAR

tTimeoutTimer(PT := tTimeout);

eState := eNextState;

CASE eState OF
	DISABLED: 	sStatusText := 'piston disabled';
	READY: 		sStatusText := 'piston ready to operate';
	BUSY: 		sStatusText := '';
	
	TIMEOUT:	sStatusText := 'piston in timeout';
				tTimeoutTimer(IN := TRUE);
				
				IF tTimeoutTimer.Q THEN
					tTimeoutTimer(IN := FALSE);
					eNextState := READY;
				END_IF

	HALTED:		sStatusText := 'piston halted';
END_CASE

METHOD M_Disable : BOOL
VAR_INPUT
END_VAR
IF eState = READY THEN
	bOutputA	:= FALSE;
	bOutputB	:= FALSE;

	bEnabled	:= FALSE;
	eNextState	:= DISABLED;
END_IF
END_METHOD

METHOD M_Enable : BOOL
VAR_INPUT
END_VAR
IF eState = DISABLED THEN
	bEnabled	:= TRUE;
	eNextState	:= READY;
END_IF
END_METHOD

METHOD M_Extend : BOOL
VAR_INPUT
END_VAR
IF eState = READY OR eState = BUSY THEN
	bOutputA	:= TRUE;
	bOutputB	:= FALSE;
END_IF
END_METHOD

METHOD M_Halt : BOOL
VAR_INPUT
END_VAR
IF eState <> HALTED AND eState <> DISABLED THEN
	bLastOutputA	:= bOutputA;
	bLastOutputB	:= bOutputB;
	M_Hold();
	eLastState 		:= eState;
	eNextState		:= HALTED;
END_IF
END_METHOD

METHOD M_Hold : BOOL
VAR_INPUT
END_VAR
IF eState = READY OR eState = BUSY THEN
	bOutputA	:= FALSE;
	bOutputB	:= FALSE;
	eNextState	:= TIMEOUT;
END_IF
END_METHOD

METHOD M_Resume : BOOL
VAR_INPUT
END_VAR
IF eState = HALTED THEN
	bOutputA	:= bLastOutputA;
	bOutputB	:= bLastOutputB;
	eNextState	:= eLastState;
END_IF
END_METHOD

METHOD M_Retract : BOOL
VAR_INPUT
END_VAR
IF eState = READY OR eState = BUSY THEN
	bOutputA	:= FALSE;
	bOutputB	:= TRUE;
END_IF
END_METHOD

END_FUNCTION_BLOCK

// ---- POUs/deprecated/FB_Module_ToolHolder_Old.TcPOU
FUNCTION_BLOCK FB_Module_ToolHolder_Old IMPLEMENTS I_Module
VAR_INPUT
	bEnable					: BOOL;
	bToolRotationBtn		: BOOL;
END_VAR
VAR_IN_OUT
	bToolRotationBtnLight	: BOOL;
END_VAR
VAR
	Components			: ARRAY [0..5] OF I_Component;
	
	fbACmotor			: FB_Component_ACmotor;
	
	fbToolHolderLock	: FB_Component_SingleValve;
	fbReedLock			: FB_Component_ReedSwitch;
	fbReedUnlock		: FB_Component_ReedSwitch;
	
	fbIndexBit1			: FB_Component_InductiveSensor;
	fbIndexBit2			: FB_Component_InductiveSensor;
	idx					: INT;
	bDir				: BOOL; // placeholder because this motor is single direction
	bToolRotating		: BOOL;
END_VAR

IF bEnable THEN
	fbACmotor(
		bDeviceActive 	:= GVL.bLenze1Relay,
		sName			:= 'AC motor holder',
		bEnable			:= TRUE,
		bE1jog1			:= GVL.bLenze2JogBit1,
		bE2jog2			:= GVL.bLenze2JogBit2,
		bE3DCbrake		:= GVL.bLenze2njectionBrake,
		eE4Direction	:= bDir);
		
	fbToolHolderLock(
		sName 	:= 'Holder Lock',
		bEnable := TRUE,
		bOutput := GVL.bUnlockToolHolder);
		
	fbReedLock(
		bRawSignal	:= GVL.bToolHolderUnlocked,
		tDebounce	:= T#5MS,
		tTimeout	:= T#0S,
		sName		:= 'holder locked reed',
		bEnable		:= TRUE);
		
	fbReedUnlock(
		bRawSignal	:= GVL.bToolHolderLocked,
		tDebounce	:= T#5MS,
		tTimeout	:= T#0S,
		sName		:= 'holder unlocked reed',
		bEnable		:= TRUE);
		
	fbIndexBit1(bRawSignal := GVL.bToolHolderIndexBit1,
		tDebounce 	:= T#5MS,
		tTimeout	:= T#0S,
		sName		:= 'holder index 1',
		bEnable		:= TRUE);
		
	fbIndexBit2(bRawSignal := GVL.bToolHolderIndexBit2,
		tDebounce 	:= T#5MS,
		tTimeout	:= T#0S,
		sName		:= 'holder index 2',
		bEnable		:= TRUE);
		
	Components[0] 	:= fbACmotor;
	Components[1] 	:= fbToolHolderLock;
	Components[2] 	:= fbReedLock;
	Components[3] 	:= fbReedUnlock;
	Components[4] 	:= fbIndexBit1;
	Components[5] 	:= fbIndexBit2;
	
	FOR idx := 0 TO 5 DO
    	Components[idx].M_Start();
	END_FOR;
	
	IF bToolRotationBtn THEN
		bToolRotating := TRUE;
	END_IF
	
	IF bToolRotating THEN
		bToolRotationBtnLight := TRUE;
		bToolRotating := NOT M_Switch();
	ELSE
		bToolRotationBtnLight := FALSE;
	END_IF
END_IF

METHOD M_Halt : BOOL
VAR_INPUT
END_VAR
END_METHOD

METHOD M_Lock : BOOL
VAR_INPUT
END_VAR

VAR
	eState: INT;
END_VAR
IF bEnable AND fbACmotor.eState <> E_State.BUSY THEN 
		fbToolHolderLock.M_Retract();
END_IF;
END_METHOD

METHOD M_Start : BOOL
VAR_INPUT
END_VAR
END_METHOD

METHOD M_Stop : BOOL
VAR_INPUT
END_VAR
END_METHOD

METHOD M_Switch : BOOL
VAR_INPUT
END_VAR

VAR
	tTrigger1 	: R_TRIG;
	tTrigger2 	: R_TRIG;
END_VAR
IF bEnable AND fbReedUnlock.bSensorActive THEN	
	tTrigger1(CLK := fbIndexBit1.bRisingEdge);					// triggers to detect rising edge of index bits
	tTrigger2(CLK := fbIndexBit2.bRisingEdge);
	
	fbACmotor.M_SetFreq(Frequency := E_LenzeJogFreq.F3);		// when no index bit has triggered, high speed
	
	IF tTrigger1.Q THEN											// when first index is triggered, switch to lowest speed
		fbACmotor.M_SetFreq(Frequency := E_LenzeJogFreq.F1);
	END_IF
	
	IF tTrigger2.Q THEN											// when last index bit has triggered, turn of motor
		fbACmotor.M_SetFreq(Frequency := E_LenzeJogFreq.FOFF);
		IF fbACmotor.eState <> E_State.BUSY THEN		// if motor is off, lock plate and signal operation done
			M_lock();
			M_Switch := TRUE;
		END_IF;
	END_IF
ELSE
	M_Unlock();													// unlock plate of locked and reset edges for detecting indexes
	fbIndexBit1.M_ResetEdge();
	fbIndexBit2.M_ResetEdge();
END_IF
END_METHOD

METHOD M_Unlock : BOOL
VAR_INPUT
END_VAR
IF bEnable AND fbACmotor.eState <> E_State.BUSY THEN 
		fbToolHolderLock.M_Extend();
END_IF;
END_METHOD

END_FUNCTION_BLOCK

// ---- POUs/FB_Components/FB_Component_DualValveGuarded.TcPOU
FUNCTION_BLOCK FB_Component_DualValveGuarded IMPLEMENTS I_Component
VAR_INPUT
	sName			: STRING[50];
	tTimeout		: TIME := T#0S;
END_VAR

VAR_IN_OUT
	bSensExtended	: BOOL;
	bSensRetracted	: BOOL;
	bOutputA		: BOOL;
	bOutputB		: BOOL;
END_VAR

VAR_OUTPUT
	bEnabled     	: BOOL;
	eState			: E_State := E_State.DISABLED;
	eNextState		: E_State := E_State.DISABLED;
	sStatusText 	: STRING[100];
	
	bIsExtended		: BOOL;
	bIsRetracted	: BOOL;
END_VAR

VAR
	bRetracting		: BOOL;
	bExtending		: BOOL;
	tTimeoutTimer	: TON;
	
	bLastOutputA	: BOOL;
	bLastOutputB	: BOOL;
	eLastState		: E_State;
	
	Components		: ARRAY [0..2] OF I_Component;
	
	fbPiston		: FB_Component_DualValve;
	fbReedExtended	: FB_Component_ReedSwitch;
	fbReedRetracted	: FB_Component_ReedSwitch;
END_VAR

VAR CONSTANT
	DISABLED		: E_State := E_State.DISABLED;
	READY			: E_State := E_State.READY;
	BUSY			: E_State := E_State.BUSY;
	DONE			: E_State := E_State.DONE;
	HALTED			: E_State := E_State.HALTED;
	TIMEOUT			: E_State := E_State.TIMEOUT;
END_VAR

tTimeoutTimer(PT := tTimeout);

fbPiston(sName := '', tTimeout 	:= T#0S, bOutputA := bOutputA, bOutputB := bOutputB);
fbReedExtended(sName := '', bRawSignal 	:= bSensExtended, tTimeout := T#0S);
fbReedRetracted(sName := '', bRawSignal 	:= bSensRetracted, tTimeout := T#0S);

Components[0] := fbPiston;
Components[1] := fbReedExtended;
Components[2] := fbReedRetracted;

bIsExtended		:= fbReedExtended.bSensorActive;
bIsRetracted	:= fbReedRetracted.bSensorActive;

eState := eNextState;

CASE eState OF
	DISABLED: 	sStatusText := 'piston disabled';
	READY: 		sStatusText :=  CONCAT(CONCAT(SEL(bIsExtended = TRUE, '', 'piston extended and '),SEL(bIsRetracted = TRUE, '', 'piston retracted and ')), 'ready to operate');
	
	BUSY: 		IF bExtending THEN
					sStatusText := 'piston extending';
					IF fbReedExtended.bSensorActive THEN
						fbPiston.M_Hold();
						eNextState := TIMEOUT;
					ELSE
						fbPiston.M_Extend();
					END_IF
				END_IF
				IF bRetracting THEN
					sStatusText := 'piston retracting';
					IF fbReedRetracted.bSensorActive THEN
						fbPiston.M_Hold();
						eNextState := TIMEOUT;
					ELSE
						fbPiston.M_Retract();
					END_IF
				END_IF
			
	TIMEOUT:	sStatusText := 'piston in timeout';
				bExtending  := FALSE;
				bRetracting := FALSE;
				tTimeoutTimer(IN := TRUE);
				
				IF tTimeoutTimer.Q THEN
					tTimeoutTimer(IN := FALSE);
					eNextState := E_State.READY;
				END_IF
				
	HALTED:		sStatusText := 'piston halted';
END_CASE

{warning 'add method implementation '}
METHOD M_Disable : BOOL
VAR
	idx	: INT := 0;
END_VAR
IF eState = READY THEN
	bEnabled	:= FALSE;
	eNextState	:= DISABLED;
	
	FOR idx := 0 TO 2 DO
    	Components[idx].M_Disable();
	END_FOR;
END_IF
END_METHOD

{warning 'add method implementation '}
METHOD M_Enable : BOOL

VAR
	idx: INT;
END_VAR
IF eState = DISABLED THEN
	bEnabled	:= TRUE;
	eNextState	:= READY;
	
	FOR idx := 0 TO 2 DO
    	Components[idx].M_Enable();
	END_FOR;
END_IF
END_METHOD

METHOD M_Extend : BOOL
VAR_INPUT
END_VAR
IF eState = READY AND NOT fbReedExtended.bSensorActive THEN
	bExtending 	:= TRUE;
	eNextState	:= BUSY;
END_IF
END_METHOD

{warning 'add method implementation '}
METHOD M_Halt : BOOL

VAR
	idx: INT;
END_VAR
IF eState <> HALTED AND eState <> DISABLED THEN
	eLastState 		:= eState;
	eNextState		:= HALTED;
	
	FOR idx := 0 TO 2 DO
		Components[idx].M_Halt();
	END_FOR;
END_IF
END_METHOD

{warning 'add method implementation '}
METHOD M_Resume : BOOL

VAR
	idx: INT;
END_VAR
IF eState = HALTED THEN
	eNextState	:= eLastState;
	bOutputA 	:= bLastOutputA;
	bOutputB 	:= bLastOutputB;
	FOR idx := 0 TO 2 DO
		Components[idx].M_Resume();
	END_FOR;
END_IF
END_METHOD

METHOD M_Retract : BOOL
VAR_INPUT
END_VAR
IF eState = READY AND NOT fbReedRetracted.bSensorActive  THEN
	bRetracting	:= TRUE;
	eNextState	:= BUSY;
END_IF
END_METHOD

END_FUNCTION_BLOCK

// ---- POUs/FB_Components/FB_Component_Servo.TcPOU
FUNCTION_BLOCK FB_Component_Servo IMPLEMENTS I_Component
VAR_INPUT
	sName				: STRING[50];			
	tTimeout			: TIME := T#0MS;
	
	uMaxRPMservo		: INT;		// value set in servo drive ( == RPM before gears!!)
	rGearRatio			: REAL;
END_VAR

VAR_IN_OUT
	bRTO				: BOOL;
	bEnableDrive		: BOOL;
	bResetDrive			: BOOL;
	uAnalogOut			: INT;
	
	(*bSetCounterDone		: BOOL;
	dCount				: DINT;
	bSetCounter			: BOOL;
	dSetCounterValue	: DINT;*)
END_VAR

VAR_OUTPUT
	
	bEnabled			: BOOL;
	eState				: E_State 				:= E_State.DISABLED;
	eServoState			: E_ServoStateMachine 	:= E_ServoStateMachine.IDLE;
	sStatusText 		: STRING[100];
END_VAR

VAR
	tTimeoutTimer		: TON;
	eLastState			: E_State;
	
	uInitialRPM			: INT;
	uTargetRPM			: INT;
	uCurrRPM			: INT;
	uSetRPM				: INT;
	uRPMlimit			: INT := 0;
	uAcceleration		: INT := 0;		// RPM/s
	bDirection			: BOOL;			// FALSE = CW, TRUE = CCW
	tAccelerationTimer	: TON;
END_VAR

VAR CONSTANT
	DISABLED			: E_State := E_State.DISABLED;
	READY				: E_State := E_State.READY;
	BUSY				: E_State := E_State.BUSY;
	DONE				: E_State := E_State.DONE;
	HALTED				: E_State := E_State.HALTED;
	TIMEOUT				: E_State := E_State.TIMEOUT;
	
	IDLE       			: E_ServoStateMachine := E_ServoStateMachine.IDLE;
	HOMING     			: E_ServoStateMachine := E_ServoStateMachine.HOMING;
	HOMED      			: E_ServoStateMachine := E_ServoStateMachine.HOMED;
	RAMPUP     			: E_ServoStateMachine := E_ServoStateMachine.RAMPUP;
	HOLD       			: E_ServoStateMachine := E_ServoStateMachine.HOLD;
	RAMPDOWN   			: E_ServoStateMachine := E_ServoStateMachine.RAMPDOWN;
	FAULT      			: E_ServoStateMachine := E_ServoStateMachine.FAULT;
END_VAR

tTimeoutTimer.PT		:= tTimeout;
tAccelerationTimer.PT 	:= T#30M;

uCurrRPM := REAL_TO_INT((((INT_TO_REAL(ABS(uAnalogOut))/32767)) * uMaxRPMservo) / rGearRatio);

CASE eState OF
	DISABLED: 	sStatusText := 'servo is disabled';
	READY: 		sStatusText := 'servo ready to operate';
	BUSY: 		sStatusText := 'servo operating';
				CASE eServoState OF
					IDLE:
						eServoState := IDLE;
					RAMPUP:
						IF NOT bRTO THEN
							eServoState := FAULT;
						END_IF
						tAccelerationTimer(IN := TRUE);
						IF uCurrRPM = uTargetRPM THEN
							eServoState := HOLD;
						ELSE
							uSetRPM 	:= M_CalculateRPM(	uTargetRPM 		:= uTargetRPM, 
															uInitialRPM 	:= uInitialRPM, 
															rElapsedTime 	:= tAccelerationTimer.ET);
							uAnalogOut 	:= REAL_TO_INT(((uSetRPM * rGearRatio) / uMaxRPMservo) * 32767);
						END_IF
					HOLD:
						IF NOT bRTO THEN
							eServoState := FAULT;
						END_IF
						IF uAnalogOut = 0 THEN
							eServoState := IDLE;
							eState 		:= READY;
						END_IF
					RAMPDOWN:
						IF NOT bRTO THEN
							eServoState := FAULT;
						END_IF
						tAccelerationTimer(IN := TRUE);
						IF uCurrRPM = uTargetRPM THEN
							eServoState := HOLD;
						ELSE
							uSetRPM 	:= M_CalculateRPM(	uTargetRPM 		:= uTargetRPM, 
															uInitialRPM 	:= uInitialRPM, 
															rElapsedTime 	:= tAccelerationTimer.ET);
							uAnalogOut 	:= REAL_TO_INT(((uSetRPM * rGearRatio) / uMaxRPMservo) * 32767);
						END_IF
					FAULT:
						IF bEnableDrive AND NOT bRTO THEN
							bResetDrive := TRUE;
							sStatusText := 'please reset servo drive';
						ELSE
							bResetDrive := FALSE;
							M_SetTargetRPM(RPM := uTargetRPM);
						END_IF
				END_CASE
	TIMEOUT:	sStatusText := '';
	DONE:		sStatusText := '';
	HALTED:		sStatusText := '';
				uAnalogOut 	:= 0;
END_CASE

METHOD M_CalculateRPM : INT
VAR_INPUT
	uTargetRPM  	: INT;
	uInitialRPM		: INT;
	rElapsedTime	: TIME;
END_VAR

VAR
	uRPMdiff		: INT; // rpm to add to initial rpm
END_VAR
uRPMdiff := REAL_TO_INT((TIME_TO_REAL(rElapsedTime) / 1000) * uAcceleration);

CASE eServoState OF
	RAMPUP:
		M_CalculateRPM := SEL((uInitialRPM + uRPMdiff) >= uTargetRPM, (uInitialRPM + uRPMdiff), uTargetRPM);
	RAMPDOWN:
		M_CalculateRPM := SEL((uInitialRPM - uRPMdiff) <= uTargetRPM, (uInitialRPM - uRPMdiff), uTargetRPM);
END_CASE
END_METHOD

{warning 'add method implementation '}
METHOD M_Disable : BOOL
IF eState = DONE OR eState = READY THEN
	bEnabled	:= FALSE;
	bEnableDrive:= FALSE;
	eState		:= DISABLED;
END_IF
END_METHOD

{warning 'add method implementation '}
METHOD M_Enable : BOOL
IF eState = DISABLED THEN
	bEnabled	:= TRUE;
	bEnableDrive:= TRUE;
	eState 		:= READY;
END_IF
END_METHOD

{warning 'add method implementation '}
METHOD M_Halt : BOOL
eLastState 	:= eState;
eState 		:= HALTED;

uAnalogOut	:= 0;
eServoState := FAULT;
tAccelerationTimer(IN := FALSE);
END_METHOD

{warning 'add method implementation '}
METHOD M_Resume : BOOL
CASE eState OF
	HALTED:		eState := eLastState;
				M_SetTargetRPM(RPM := uTargetRPM);
	DONE:		eState := READY;
END_CASE
END_METHOD

METHOD M_SetAcceleration : BOOL
VAR_INPUT
	uRPMperSec : INT;
END_VAR
uAcceleration := SEL(uRPMperSec >= 500, uRPMperSec, 500);
END_METHOD

METHOD M_SetRPMlimit : BOOL
VAR_INPUT
	RPM 				: INT;
END_VAR

VAR
	uMaxRPMafterGears	: INT;
END_VAR
uMaxRPMafterGears 	:= REAL_TO_INT(INT_TO_REAL(uMaxRPMservo) / rGearRatio);
uRPMlimit 			:= SEL(RPM >= uMaxRPMafterGears, RPM, uMaxRPMafterGears);
END_METHOD

METHOD M_SetTargetRPM : BOOL
VAR_INPUT
	RPM : INT;
END_VAR
IF eState = READY OR eState = BUSY THEN
	tAccelerationTimer(IN := FALSE);	// reset the timer
	uTargetRPM 	:= SEL(RPM >= uRPMlimit, RPM, uRPMlimit);
	uInitialRPM	:= uCurrRPM;
	
	IF uTargetRPM > uCurrRPM THEN
		eState 		:= BUSY;
		eServoState := RAMPUP;
	ELSIF uTargetRPM < uCurrRPM THEN
		eState 		:= BUSY;
		eServoState := RAMPDOWN;
	ELSIF uTargetRPM = 0 AND uCurrRPM = 0 THEN
		eState 		:= READY;
		eServoState := IDLE;
	ELSE
		eState 		:= BUSY;
		eServoState := HOLD;
	END_IF
END_IF;
END_METHOD

{warning 'add method implementation '}
METHOD M_Stop : BOOL
IF eState <> BUSY OR eState <> HALTED OR eState <> TIMEOUT THEN
	// reset all values to 0
	eState := DONE;
END_IF
END_METHOD

END_FUNCTION_BLOCK

// ---- POUs/FB_Components/FB_Component_SingleValveGuarded.TcPOU
FUNCTION_BLOCK FB_Component_SingleValveGuarded IMPLEMENTS I_Component
VAR_INPUT
	sName			: STRING[50];
	tTimeout		: TIME := T#0S;
END_VAR

VAR_IN_OUT
	bSensExtended	: BOOL;
	bSensRetracted	: BOOL;
	bOutput			: BOOL;
END_VAR

VAR_OUTPUT
	bEnabled     	: BOOL;
	eState			: E_State := E_State.DISABLED;
	eNextState		: E_State := E_State.DISABLED;
	sStatusText 	: STRING[100];
	
	bIsExtended		: BOOL;
	bIsRetracted	: BOOL;
END_VAR

VAR
	bTest			: BOOL;
	bRetracting		: BOOL;
	bExtending		: BOOL;
	tTimeoutTimer	: TON;

	eLastState		: E_State;
	
	Components		: ARRAY [0..2] OF I_Component;
	
	fbPiston		: FB_Component_SingleValve;
	fbReedExtended	: FB_Component_ReedSwitch;
	fbReedRetracted	: FB_Component_ReedSwitch;
END_VAR

VAR CONSTANT
	DISABLED		: E_State := E_State.DISABLED;
	READY			: E_State := E_State.READY;
	BUSY			: E_State := E_State.BUSY;
	DONE			: E_State := E_State.DONE;
	HALTED			: E_State := E_State.HALTED;
	TIMEOUT			: E_State := E_State.TIMEOUT;
END_VAR

tTimeoutTimer(PT := tTimeout);

fbPiston(sName := '', tTimeout 	:= T#0S, bOutput := bOutput);
fbReedExtended(sName := '', bRawSignal 	:= bSensExtended, tTimeout := T#0S);
fbReedRetracted(sName := '', bRawSignal 	:= bSensRetracted, tTimeout := T#0S);

Components[0] := fbPiston;
Components[1] := fbReedExtended;
Components[2] := fbReedRetracted;

bIsExtended		:= fbReedExtended.bSensorActive;
bIsRetracted	:= fbReedRetracted.bSensorActive;

eState := eNextState;

CASE eState OF
	DISABLED: 	sStatusText := 'piston disabled';
	READY: 		sStatusText :=  CONCAT(CONCAT(SEL(bIsExtended = TRUE, '', 'piston extended and '),SEL(bIsRetracted = TRUE, '', 'piston retracted and ')), 'ready to operate');
	
	BUSY: 		IF bExtending THEN
					sStatusText := 'piston extending';
					IF fbReedExtended.bSensorActive THEN
						eNextState := TIMEOUT;
					ELSE
						fbPiston.M_Extend();
					END_IF
				END_IF
				IF bRetracting THEN
					sStatusText := 'piston retracting';
					IF fbReedRetracted.bSensorActive THEN
						eNextState := TIMEOUT;
					ELSE
						fbPiston.M_Retract();
					END_IF
				END_IF
			
	TIMEOUT:	sStatusText := 'piston in timeout';
				bExtending  := FALSE;
				bRetracting := FALSE;
				tTimeoutTimer(IN := TRUE);
				
				IF tTimeoutTimer.Q THEN
					tTimeoutTimer(IN := FALSE);
					eNextState := READY;
				END_IF
				
	HALTED:		sStatusText := 'piston halted';
END_CASE

{warning 'add method implementation '}
METHOD M_Disable : BOOL
VAR
	idx	: INT := 0;
END_VAR
IF eState = READY THEN
	bEnabled	:= FALSE;
	eNextState	:= DISABLED;
	
	FOR idx := 0 TO 2 DO
    	Components[idx].M_Disable();
	END_FOR;
END_IF
END_METHOD

{warning 'add method implementation '}
METHOD M_Enable : BOOL

VAR
	idx: INT;
END_VAR
IF eState = DISABLED THEN
	bEnabled	:= TRUE;
	eNextState	:= READY;
	
	FOR idx := 0 TO 2 DO
    	Components[idx].M_Enable();
	END_FOR;
END_IF
END_METHOD

METHOD M_Extend : BOOL
VAR_INPUT
END_VAR
IF eState = READY AND NOT fbReedExtended.bSensorActive THEN
	bExtending 	:= TRUE;
	eNextState	:= BUSY;
END_IF
END_METHOD

{warning 'add method implementation '}
METHOD M_Halt : BOOL

VAR
	idx: INT;
END_VAR
IF eState <> HALTED AND eState <> DISABLED THEN
	eLastState 		:= eState;
	eNextState		:= HALTED;
	FOR idx := 0 TO 2 DO
		Components[idx].M_Halt();
	END_FOR;
END_IF
END_METHOD

{warning 'add method implementation '}
METHOD M_Resume : BOOL

VAR
	idx: INT;
END_VAR
IF eState = HALTED THEN
	eNextState := eLastState;
	FOR idx := 0 TO 2 DO
		Components[idx].M_Resume();
	END_FOR;
END_IF
END_METHOD

METHOD M_Retract : BOOL
VAR_INPUT
END_VAR
IF eState = READY AND NOT fbReedRetracted.bSensorActive  THEN
	bRetracting	:= TRUE;
	eNextState	:= BUSY;
END_IF
END_METHOD

END_FUNCTION_BLOCK

// ---- POUs/FB_Components/FB_Component_4posArm.TcPOU
FUNCTION_BLOCK FB_Component_4posArm IMPLEMENTS I_Component
VAR_INPUT
	sName			: STRING[50];
	tTimeout		: TIME := T#0S;
END_VAR

VAR_IN_OUT
END_VAR

VAR_OUTPUT
	bEnabled     	: BOOL;
	eState			: E_State := E_State.DISABLED;
	eNextState		: E_State := E_State.DISABLED;
	nCurrentIndex	: INT;
	sStatusText 	: STRING[100];
END_VAR

VAR
	eLastState		: E_State;
	tTimeoutTimer	: TON;
	Components		: ARRAY [0..4] OF I_Component;	
	
	fbPiston		: FB_Component_DualValve;
	fbIndex1		: FB_Component_ReedSwitch;
	fbIndex2		: FB_Component_ReedSwitch;
	fbIndex3		: FB_Component_ReedSwitch;
	fbIndex4		: FB_Component_ReedSwitch;
	
	nTargetIndex	: INT;
END_VAR

VAR CONSTANT
	DISABLED		: E_State := E_State.DISABLED;
	READY			: E_State := E_State.READY;
	BUSY			: E_State := E_State.BUSY;
	HALTED			: E_State := E_State.HALTED;
	TIMEOUT			: E_State := E_State.TIMEOUT;
END_VAR

tTimeoutTimer(PT := tTimeout);

fbPiston(sName := 'piston for 4 pos arm', bOutputA := GVL.bExtendWireHolder, bOutputB := GVL.bRetractWireHolder);
fbIndex1(sName := '4pos arm index bit 1', bRawSignal := GVL.bWireHolderPos1);
fbIndex2(sName := '4pos arm index bit 2', bRawSignal := GVL.bWireHolderPos2);
fbIndex3(sName := '4pos arm index bit 3', bRawSignal := GVL.bWireHolderPos3);
fbIndex4(sName := '4pos arm index bit 4', bRawSignal := GVL.bWireHolderPos4);

Components[0] := fbPiston;
Components[1] := fbIndex1;
Components[2] := fbIndex2;
Components[3] := fbIndex3;
Components[4] := fbIndex4;

IF fbIndex1.bSensorActive THEN
	nCurrentIndex := 1;
ELSIF fbIndex2.bSensorActive THEN
	nCurrentIndex := 2;
ELSIF fbIndex3.bSensorActive THEN
	nCurrentIndex := 3;
ELSIF fbIndex4.bSensorActive THEN
	nCurrentIndex := 4;
END_IF

eState := eNextState;

// TEST IF WHEN HALTED INBETWEEN INDEXES IF IT FIXES ITSELF. IT SHOULD

CASE eState OF
	DISABLED: 	sStatusText := '4 pos arm disabled';
	READY: 		sStatusText := CONCAT('4 pos arm is ready to operate and at index: ', INT_TO_STRING(nCurrentIndex));
	
	BUSY: 		IF nTargetIndex > nCurrentIndex THEN
					fbPiston.M_Extend();
					sStatusText := '4 pos arm is extending';
				ELSIF	nTargetIndex < nCurrentIndex THEN
					fbPiston.M_Retract();
					sStatusText := '4 pos arm is retracting';
				ELSE
					fbPiston.M_Hold();
					eNextState := TIMEOUT;
				END_IF
				
	TIMEOUT:	sStatusText := '4 pos arm is in timeout';
				tTimeoutTimer(IN := TRUE);
				
				IF tTimeoutTimer.Q THEN
					tTimeoutTimer(IN := FALSE);
					eNextState := READY;
				END_IF
				
	HALTED:		sStatusText := '4 pos arm is halted';
END_CASE

{warning 'add method implementation '}
METHOD M_Disable : BOOL

VAR
	idx: INT;
END_VAR
IF eState = READY THEN
	bEnabled	:= FALSE;
	eNextState	:= DISABLED;
	
	FOR idx := 0 TO 4 DO
    	Components[idx].M_Disable();
	END_FOR;
END_IF
END_METHOD

{warning 'add method implementation '}
METHOD M_Enable : BOOL

VAR
	idx: INT;
END_VAR
IF eState = DISABLED THEN
	bEnabled	:= TRUE;
	eNextState	:= READY;
	
	FOR idx := 0 TO 4 DO
    	Components[idx].M_Enable();
	END_FOR;
END_IF
END_METHOD

{warning 'add method implementation '}
METHOD M_Halt : BOOL

VAR
	idx: INT;
END_VAR
IF eState <> HALTED AND eState <> DISABLED THEN
	eLastState 		:= eState;
	eNextState		:= HALTED;
	FOR idx := 0 TO 4 DO
		Components[idx].M_Halt();
	END_FOR;
END_IF
END_METHOD

{warning 'add method implementation '}
METHOD M_Resume : BOOL

VAR
	idx: INT;
END_VAR
IF eState = HALTED THEN
	eNextState := eLastState;
	FOR idx := 0 TO 4 DO
		Components[idx].M_Resume();
	END_FOR;
END_IF
END_METHOD

METHOD M_SetTargetIndex : BOOL
VAR_INPUT
	index : INT;
END_VAR
IF eState = READY OR eState = BUSY THEN
	nTargetIndex 	:= index;
	eNextState 		:= BUSY;
END_IF
END_METHOD

END_FUNCTION_BLOCK

// ---- POUs/FB_Component_ServoMotor.TcPOU
FUNCTION_BLOCK FB_Component_ServoMotor IMPLEMENTS I_Component
VAR_INPUT
	bEnable				: BOOL;	

	bHomingSensor		: BOOL;
	bHomingSpeed		: INT;
	uMaxRPM				: INT;
	bSetCounterDone		: BOOL;
	rGearRatio			: REAL;
END_VAR
VAR_IN_OUT
	dCountServo			: DINT;
	bSetCounter			: BOOL;
	dSetCounterValue	: DINT;
	bEnableDrive		: BOOL;
	uAnalogOut			: INT;
END_VAR
VAR_OUTPUT
	uCurrRPM			: INT;
END_VAR
VAR
	tHomeTrig			: F_TRIG;
	bHomeTriggered		: BOOL;
END_VAR

(*

aOutServo2						AT %Q*	: INT;	// term 18.1

bSetCounterDoneServo2			AT %I*	: BOOL;
dCountServo2					AT %I*	: DINT;

dSetCounterServo2				AT %Q*	: BOOL;
dSetCounterValueServo2			AT %Q*	: DINT;
*)

IF bEnable THEN
	uCurrRPM := REAL_TO_INT((((INT_TO_REAL(ABS(uAnalogOut))/32767)) * uMaxRPM) / rGearRatio);
ELSE
	bEnableDrive := FALSE;
	uAnalogOut	 := 0;
	uCurrRPM	 := 0;
END_IF

METHOD M_DisableDrive : BOOL
VAR_INPUT
END_VAR
IF bEnable THEN
	bEnableDrive := FALSE;
END_IF
END_METHOD

METHOD M_EnableDrive : BOOL
VAR_INPUT
END_VAR
IF bEnable THEN
	bEnableDrive := TRUE;
END_IF
END_METHOD

METHOD M_Goto : BOOL
VAR_INPUT
	dTarget			: DINT;
	uSpeed			: INT;
	uMargin			: INT;
END_VAR
VAR
END_VAR
IF bEnable THEN
	// safety
	IF uSpeed > 5 THEN
		RETURN;
	END_IF
	
	IF dTarget > dCountServo THEN
		M_EnableDrive();
		IF ABS(dTarget - dCountServo) > uMargin THEN
			M_SetSpeed(uSpeed);
		ELSE
			M_SetSpeed(0.5);
		END_IF
	ELSIF  dTarget < dCountServo THEN
		M_EnableDrive();
		IF ABS(dCountServo - dTarget)  > uMargin THEN
			M_SetSpeed(-uSpeed);
		ELSE
			M_SetSpeed(-0.5);
		END_IF
	ELSE
		M_EnableDrive();
		M_SetSpeed(0);
		M_Goto := TRUE;
	END_IF
END_IF
END_METHOD

{warning 'add method implementation '}
METHOD M_Halt : BOOL
END_METHOD

METHOD M_SetCounter : BOOL
VAR_INPUT
	dCount : DINT;
END_VAR
IF bEnable THEN
	IF bSetCounterDone THEN
		bSetCounter			:= FALSE;
		M_SetCounter 		:= TRUE;
	ELSE
		dSetCounterValue 	:= dCount;
		bSetCounter			:= TRUE;
	END_IF
END_IF
END_METHOD

METHOD M_SetSpeed : BOOL
VAR_INPUT
	uSpeed	: REAL;
END_VAR
IF bEnable THEN
	uAnalogOut := LIMIT(-32767, REAL_TO_INT(uSpeed * 327.67), 32767);
END_IF
END_METHOD

{warning 'add method implementation '}
METHOD M_Start : BOOL
END_METHOD

{warning 'add method implementation '}
METHOD M_Stop : BOOL
END_METHOD

END_FUNCTION_BLOCK

// ---- POUs/FB_Modules/FB_Module_CoilHolder.TcPOU
FUNCTION_BLOCK FB_Module_CoilHolder IMPLEMENTS I_Module
VAR_INPUT
	sName			: STRING[50];
	tTimeout		: TIME := T#0S;
END_VAR

VAR_IN_OUT
END_VAR

VAR_OUTPUT
	bEnabled     	: BOOL;
	eState			: E_State := E_State.DISABLED;
	eNextState		: E_State := E_State.DISABLED;
	nCurrentIndex	: INT;
	sStatusText 	: STRING[100];
END_VAR

VAR
	eLastState		: E_State;
	tTimeoutTimer	: TON;
	Components		: ARRAY [0..7] OF I_Component;

	fbMotor			: FB_Component_ACmotor;
	fbPistonLock	: FB_Component_SingleValveGuarded;	
	fbIndexReadyBit	: FB_Component_InductiveSensor;
	fbIndexBit1		: FB_Component_InductiveSensor;
	fbIndexBit2		: FB_Component_InductiveSensor;
	fbIndexBit3		: FB_Component_InductiveSensor;
	fbIndexBit4		: FB_Component_InductiveSensor;
	fbIndexBit5		: FB_Component_InductiveSensor;
	
	nTargetIndex	: INT;
	cwSteps			: INT;
	ccwSteps		: INT;
	shortestDistance: INT;
END_VAR

VAR CONSTANT
	DISABLED		: E_State := E_State.DISABLED;
	READY			: E_State := E_State.READY;
	BUSY			: E_State := E_State.BUSY;
	HALTED			: E_State := E_State.HALTED;
	TIMEOUT			: E_State := E_State.TIMEOUT;
	
	CW				: E_RotationDirection := E_RotationDirection.CW;
	CCW				: E_RotationDirection := E_RotationDirection.CCW;
	
	FOFF			: E_LenzeJogFreq := E_LenzeJogFreq.FOFF;
	F1				: E_LenzeJogFreq := E_LenzeJogFreq.F1;
	F2				: E_LenzeJogFreq := E_LenzeJogFreq.F2;
	F3				: E_LenzeJogFreq := E_LenzeJogFreq.F3;
END_VAR

tTimeoutTimer(PT := tTimeout);

fbMotor(		sName := 'motor for coil holder', 
				bDeviceActive 	:= GVL.bLenze1Relay, 
				bE1jog1 		:= GVL.bLenze1JogBit1, 
				bE2jog2 		:= GVL.bLenze1JogBit2, 
				bE3DCbrake 		:= GVL.bLenze1InjectionBrake, 
				eE4Direction	:= gvl.bLenze1Direction);
				
fbPistonLock(	sName := 'lock for coil holder',
				bSensExtended := GVL.bCoilHolderUnlocked,
				bSensRetracted := GVL.bCoilHolderLocked,
				bOutput := GVL.bUnlockCoilHolder);

fbIndexReadyBit(sName := 'index ready bit for coil holder', bRawSignal := GVL.bCoilHolderIndexReady);

fbIndexBit1(sName := 'index bit 1 for coil holder', bRawSignal := GVL.bCoilHolderIndexBit1);
fbIndexBit2(sName := 'index bit 2 for coil holder', bRawSignal := GVL.bCoilHolderIndexBit2);
fbIndexBit3(sName := 'index bit 3 for coil holder', bRawSignal := GVL.bCoilHolderIndexBit3);
fbIndexBit4(sName := 'index bit 4 for coil holder', bRawSignal := GVL.bCoilHolderIndexBit4);
fbIndexBit5(sName := 'index bit 5 for coil holder', bRawSignal := GVL.bCoilHolderIndexBit5);

Components[0] := fbMotor;
Components[1] := fbPistonLock;
Components[2] := fbIndexReadyBit; 
Components[3] := fbIndexBit1; 
Components[4] := fbIndexBit2; 
Components[5] := fbIndexBit3; 
Components[6] := fbIndexBit4; 
Components[7] := fbIndexBit5; 

IF fbIndexReadyBit.bSensorActive THEN
	nCurrentIndex := 	TO_INT(	SHL(TO_UINT(fbIndexBit5.bSensorActive), 4) OR
								SHL(TO_UINT(fbIndexBit4.bSensorActive), 3) OR
								SHL(TO_UINT(fbIndexBit3.bSensorActive), 2) OR
								SHL(TO_UINT(fbIndexBit2.bSensorActive), 1) OR
						   		   (TO_UINT(fbIndexBit1.bSensorActive)));
END_IF

CASE eState OF
	DISABLED: 	sStatusText := 'Coil holder disabled';
	READY: 		sStatusText := CONCAT('coil holder is ready to operate and at index: ', INT_TO_STRING(nCurrentIndex));
	
	BUSY: 		IF fbPistonLock.bIsExtended THEN
					IF nTargetIndex = nCurrentIndex THEN
						fbMotor.M_SetFreq(Frequency := FOFF);
						fbPistonLock.M_Retract();
						eNextState := TIMEOUT;
					ELSE
						cwSteps  := (nTargetIndex - nCurrentIndex + 24) MOD 24;
						ccwSteps := (nCurrentIndex - nTargetIndex + 24) MOD 24;
						
						IF cwSteps <= ccwSteps THEN
							fbMotor.M_SetDir(Direction := CW);
							shortestDistance := cwSteps;
						ELSE
							fbMotor.M_SetDir(Direction := CCW);	
							shortestDistance := ccwSteps;
						END_IF
						
						IF nCurrentIndex <> nTargetIndex THEN
							IF shortestDistance <= 1 THEN
								fbMotor.M_SetFreq(Frequency := F1);	
							ELSIF shortestDistance <= 2 THEN
								fbMotor.M_SetFreq(Frequency := F2);
							ELSE
								fbMotor.M_SetFreq(Frequency := F3);
							END_IF
						ELSE
							fbMotor.M_SetFreq(Frequency := FOFF);
							fbPistonLock.M_Retract();
							eNextState := TIMEOUT;
						END_IF
					END_IF
				ELSE
					fbPistonLock.M_Extend();
				END_IF
	TIMEOUT:	sStatusText := 'Coil holder is in timeout';
				tTimeoutTimer(IN := TRUE);
				
				IF tTimeoutTimer.Q THEN
					tTimeoutTimer(IN := FALSE);
					eNextState := READY;
				END_IF
	HALTED:		sStatusText := 'Coil holder halted';
END_CASE 
eState := eNextState;

{warning 'add method implementation '}
METHOD M_Disable : BOOL

VAR
	idx: INT;
END_VAR
IF eState = READY THEN
	bEnabled	:= FALSE;
	eNextState	:= DISABLED;
	
	FOR idx := 0 TO 7 DO
    	Components[idx].M_Disable();
	END_FOR;
END_IF
END_METHOD

{warning 'add method implementation '}
METHOD M_Enable : BOOL

VAR
	idx: INT;
END_VAR
IF eState = DISABLED THEN
	bEnabled	:= TRUE;
	eNextState	:= READY;
	
	FOR idx := 0 TO 7 DO
    	Components[idx].M_Enable();
	END_FOR;
END_IF
END_METHOD

{warning 'add method implementation '}
METHOD M_Halt : BOOL

VAR
	idx: INT;
END_VAR
IF eState <> HALTED AND eState <> DISABLED THEN
	eLastState 		:= eState;
	eNextState		:= HALTED;
	FOR idx := 0 TO 7 DO
		Components[idx].M_Halt();
	END_FOR;
END_IF
END_METHOD

{warning 'add method implementation '}
METHOD M_Resume : BOOL

VAR
	idx: INT;
END_VAR
IF eState = HALTED THEN
	eNextState := eLastState;
	FOR idx := 0 TO 7 DO
		Components[idx].M_Resume();
	END_FOR;
END_IF
END_METHOD

METHOD M_SetTargetIndex : BOOL
VAR_INPUT
	index : INT;
END_VAR
IF eState = READY OR eState = BUSY THEN
	nTargetIndex 	:= index;
	eNextState 		:= BUSY;
END_IF
END_METHOD

END_FUNCTION_BLOCK

// ---- POUs/FB_Modules/FB_Module_ToolHolder.TcPOU
FUNCTION_BLOCK FB_Module_ToolHolder IMPLEMENTS I_Module
VAR_INPUT
	sName					: STRING[50];
	tTimeout				: TIME := T#0S;
END_VAR

VAR_IN_OUT
END_VAR

VAR_OUTPUT
	bEnabled     	: BOOL;
	eState			: E_State := E_State.DISABLED;
	eNextState		: E_State := E_State.DISABLED;
	sStatusText 	: STRING[100];
END_VAR

VAR
	eLastState		: E_State;
	tTimeoutTimer	: TON;
	Components		: ARRAY [0..3] OF I_Component;
	
	fbACmotor			: FB_Component_ACmotor;
	fbToolHolderLock	: FB_Component_SingleValveGuarded;
	fbIndexBit1			: FB_Component_InductiveSensor;
	fbIndexBit2			: FB_Component_InductiveSensor;
	
	bDir				: BOOL;
	bToolRotating		: BOOL;
END_VAR

VAR CONSTANT
	DISABLED		: E_State := E_State.DISABLED;
	READY			: E_State := E_State.READY;
	BUSY			: E_State := E_State.BUSY;
	HALTED			: E_State := E_State.HALTED;
	TIMEOUT			: E_State := E_State.TIMEOUT;
	
	FOFF			: E_LenzeJogFreq := E_LenzeJogFreq.FOFF;
	F1				: E_LenzeJogFreq := E_LenzeJogFreq.F1;
	F2				: E_LenzeJogFreq := E_LenzeJogFreq.F2;
	F3				: E_LenzeJogFreq := E_LenzeJogFreq.F3;
END_VAR

tTimeoutTimer(PT := tTimeout);

fbACmotor(	sName 			:= 'motor for tool rotating table',
			bDeviceActive 	:= GVL.bLenze2Relay,
			bE1jog1			:= GVL.bLenze2JogBit1,
			bE2jog2			:= GVL.bLenze2JogBit2,
			bE3DCbrake		:= GVL.bLenze2njectionBrake,
			eE4Direction	:= bDir);

fbToolHolderLock( 	sName			:= 'lock for rotating table',
					bSensExtended	:= GVL.bToolHolderUnlocked,
					bSensRetracted  := GVL.bToolHolderLocked,
					bOutput			:= GVL.bUnlockToolHolder);
					
fbIndexBit1( sName := 'index bit 1 rotating table', bRawSignal := GVL.bToolHolderIndexBit1);
fbIndexBit2( sName := 'index bit 2 rotating table', bRawSignal := GVL.bToolHolderIndexBit2);

Components[0] := fbACmotor;
Components[1] := fbToolHolderLock;
Components[2] := fbIndexBit1;
Components[3] := fbIndexBit2;
			
eState := eNextState;

CASE eState OF
	DISABLED: 	sStatusText := 'Tool rotating table is disabled';
				GVL.bToolingRotationBtnLight := FALSE;
	READY: 		sStatusText := 'Tool rotating table is ready to operate';
				IF GVL.bToolingRotationBtn THEN
					eNextState := BUSY;
				END_IF
				GVL.bToolingRotationBtnLight := FALSE;
				
	BUSY: 		IF fbToolHolderLock.bIsExtended THEN
					fbACmotor.M_SetFreq(Frequency := F2);
					
					IF fbIndexBit1.bRisingEdge THEN											// when first index is triggered, switch to lowest speed
						fbACmotor.M_SetFreq(Frequency := F1);
					END_IF
					
					IF fbIndexBit2.bRisingEdge THEN											// when last index bit has triggered, turn of motor
						fbACmotor.M_SetFreq(Frequency := E_LenzeJogFreq.FOFF);
						IF fbACmotor.eState <> E_State.BUSY THEN		// if motor is off, lock plate and signal operation done
							fbToolHolderLock.M_Retract();
							eNextState := TIMEOUT;	
						END_IF;
					END_IF
				ELSE
					fbToolHolderLock.M_Extend();
					fbIndexBit1.M_ResetEdge();
					fbIndexBit2.M_ResetEdge();
				END_IF
				GVL.bToolingRotationBtnLight := TRUE;
				
	TIMEOUT:	sStatusText := 'Tool rotating table is in timeout';
				tTimeoutTimer(IN := TRUE);
				
				IF tTimeoutTimer.Q THEN
					tTimeoutTimer(IN := FALSE);
					eNextState := READY;
				END_IF
				GVL.bToolingRotationBtnLight := TRUE;
				
	HALTED:		sStatusText := 'Tool rotating table is halted';
				GVL.bToolingRotationBtnLight := FALSE;
END_CASE

{warning 'add method implementation '}
METHOD M_Disable : BOOL

VAR
	idx: INT;
END_VAR
IF eState = READY THEN
	bEnabled	:= FALSE;
	eNextState	:= DISABLED;
	
	FOR idx := 0 TO 3 DO
    	Components[idx].M_Disable();
	END_FOR;
END_IF
END_METHOD

{warning 'add method implementation '}
METHOD M_Enable : BOOL

VAR
	idx: INT;
END_VAR
IF eState = DISABLED THEN
	bEnabled	:= TRUE;
	eNextState	:= READY;
	
	FOR idx := 0 TO 3 DO
    	Components[idx].M_Enable();
	END_FOR;
END_IF
END_METHOD

{warning 'add method implementation '}
METHOD M_Halt : BOOL

VAR
	idx: INT;
END_VAR
IF eState <> HALTED AND eState <> DISABLED THEN
	eLastState 		:= eState;
	eNextState		:= HALTED;
	FOR idx := 0 TO 3 DO
		Components[idx].M_Halt();
	END_FOR;
END_IF
END_METHOD

{warning 'add method implementation '}
METHOD M_Resume : BOOL

VAR
	idx: INT;
END_VAR
IF eState = HALTED THEN
	eNextState := eLastState;
	FOR idx := 0 TO 3 DO
		Components[idx].M_Resume();
	END_FOR;
END_IF
END_METHOD

END_FUNCTION_BLOCK

// ---- POUs/FB_Modules/FB_Module_ToolHolderDoor.TcPOU
FUNCTION_BLOCK FB_Module_ToolHolderDoor IMPLEMENTS I_Module
VAR_INPUT
	sName			: STRING[50];
	tTimeout		: TIME := T#0S;
END_VAR

VAR_IN_OUT
END_VAR

VAR_OUTPUT
	bEnabled     	: BOOL;
	eState			: E_State := E_State.DISABLED;
	eNextState		: E_State := E_State.DISABLED;
	sStatusText 	: STRING[100];
	
	bDoorOpening	: BOOL;
	bDoorClosing	: BOOL;
END_VAR

VAR
	eLastState		: E_State;
	tTimeoutTimer	: TON;
	Components		: ARRAY [0..0] OF I_Component;	
	fbPiston		: FB_Component_DualValveGuarded;
END_VAR

VAR CONSTANT
	DISABLED		: E_State := E_State.DISABLED;
	READY			: E_State := E_State.READY;
	BUSY			: E_State := E_State.BUSY;
	HALTED			: E_State := E_State.HALTED;
	TIMEOUT			: E_State := E_State.TIMEOUT;
END_VAR

tTimeoutTimer(PT := tTimeout);

fbPiston(	sName 			:= 'piston for toolholder door', 
			bSensExtended 	:= GVL.bDoorToolHolderDown, 
			bSensRetracted 	:= GVL.bDoorToolHolderLock, 
			bOutputA 		:= GVL.bOpenToolCarrierDoor, 
			bOutputB 		:= GVL.bCloseToolCarrierDoor); 
			
Components[0] := fbPiston;

eState := eNextState;

CASE eState OF
	DISABLED: 	sStatusText := 'tool holder door is disabled';
	READY: 		sStatusText := 'tool holder door is ready to operate';
	BUSY: 		IF bDoorOpening THEN
					sStatusText := 'door opening';
					IF fbPiston.bIsExtended THEN
						bDoorOpening 	:= FALSE;
						eNextState 		:= TIMEOUT;
					END_IF
				ELSIF bDoorClosing THEN
					sStatusText := 'door closing';
					IF fbPiston.bIsRetracted THEN
						bDoorClosing 	:= FALSE;
						eNextState 		:= TIMEOUT;
					END_IF
				END_IF
				
	TIMEOUT:	sStatusText := 'Tool holder door is in timeout';
				tTimeoutTimer(IN := TRUE);
				
				IF tTimeoutTimer.Q THEN
					tTimeoutTimer(IN := FALSE);
					eNextState := READY;
				END_IF
				
	HALTED:		sStatusText := 'Tool holder door is halted';
END_CASE

METHOD M_Close : BOOL
VAR_INPUT
END_VAR
IF eState = READY OR eState = BUSY THEN
	eNextState 		:= BUSY;
	bDoorClosing 	:= TRUE;
	fbPiston.M_Retract();
END_IF
END_METHOD

{warning 'add method implementation '}
METHOD M_Disable : BOOL

VAR
	idx: INT;
END_VAR
IF eState = READY THEN
	bEnabled	:= FALSE;
	eNextState	:= DISABLED;
	
	FOR idx := 0 TO 0 DO
    	Components[idx].M_Disable();
	END_FOR;
END_IF
END_METHOD

{warning 'add method implementation '}
METHOD M_Enable : BOOL

VAR
	idx: INT;
END_VAR
IF eState = DISABLED THEN
	bEnabled	:= TRUE;
	eNextState	:= READY;
	
	FOR idx := 0 TO 0 DO
    	Components[idx].M_Enable();
	END_FOR;
END_IF
END_METHOD

{warning 'add method implementation '}
METHOD M_Halt : BOOL

VAR
	idx: INT;
END_VAR
IF eState <> HALTED AND eState <> DISABLED THEN
	eLastState 		:= eState;
	eNextState		:= HALTED;
	FOR idx := 0 TO 0 DO
		Components[idx].M_Halt();
	END_FOR;
END_IF
END_METHOD

METHOD M_Open : BOOL
VAR_INPUT
END_VAR
IF eState = READY OR eState = BUSY THEN
	eNextState 		:= BUSY;
	bDoorOpening 	:= TRUE;
	fbPiston.M_Extend();
END_IF
END_METHOD

{warning 'add method implementation '}
METHOD M_Resume : BOOL

VAR
	idx: INT;
END_VAR
IF eState = HALTED THEN
	eNextState := eLastState;
	FOR idx := 0 TO 0 DO
		Components[idx].M_Resume();
	END_FOR;
END_IF
END_METHOD

END_FUNCTION_BLOCK

// ---- POUs/FB_Modules/FB_Module_Winder.TcPOU
FUNCTION_BLOCK FB_Module_Winder IMPLEMENTS I_Module
VAR_INPUT
	sName			: STRING[50];
	tTimeout		: TIME := T#0S;
END_VAR

VAR_OUTPUT
	bEnabled     	: BOOL;
	eState			: E_State;
	sStatusText 	: STRING[100];
END_VAR

VAR
	fbServo		: FB_Component_Servo;
	fbSens		: FB_Component_InductiveSensor;
	
	Components	: ARRAY [0..4] OF I_Component;
	eLastState	: E_State;
	
	uTargetRev	: INT;
	uTargetRPM	: INT;
END_VAR

VAR CONSTANT
	DISABLED		: E_State := E_State.DISABLED;
	READY			: E_State := E_State.READY;
	BUSY			: E_State := E_State.BUSY;
	DONE			: E_State := E_State.DONE;
	HALTED			: E_State := E_State.HALTED;
	TIMEOUT			: E_State := E_State.TIMEOUT;
END_VAR

fbServo(	sName 			:= 'servo for winder',
			tTimeout 		:= T#0S,
			uMaxRPMservo 	:= 3000,
			rGearRatio 		:= 2.25,
			bRTO 			:= GVL.bReadyToOperate614,
			bEnableDrive 	:= GVL.b614Enable,
			bResetDrive 	:= GVL.bResetServosErrors,
			uAnalogOut 		:= GVL.aOutServo2);
			
fbServo.M_SetAcceleration(uRPMperSec := 50);
fbServo.M_SetRPMlimit(RPM := 700);
			
fbSens(		sName			:= 'homing sensor winder',
			bRawSignal		:= GVL.bCoilRotate,
			tDebounce		:= T#0MS,
			tTimeout		:= T#0MS);
			
Components[0] := fbServo;
Components[1] := fbSens;

CASE eState OF
	DISABLED: 	sStatusText := '';
	READY:		sStatusText := '';
	BUSY:		sStatusText := '';
	TIMEOUT:	sStatusText := '';
	DONE:		sStatusText := '';
	HALTED:		sStatusText := '';
END_CASE

{warning 'add method implementation '}
METHOD M_Disable : BOOL

VAR
	idx: INT;
END_VAR
IF eState = DONE OR eState = READY THEN
	bEnabled	:= FALSE;
	eState		:= DISABLED;
	
	FOR idx := 0 TO 1 DO
    	Components[idx].M_Disable();
	END_FOR;
END_IF
END_METHOD

METHOD M_Enable : BOOL

VAR
	idx: INT;
END_VAR
IF eState = DISABLED THEN
	bEnabled	:= TRUE;
	eState 		:= READY;
	
	FOR idx := 0 TO 1 DO
    	Components[idx].M_Enable();
	END_FOR;
END_IF
END_METHOD

{warning 'add method implementation '}
METHOD M_Halt : BOOL

VAR
	idx: INT;
END_VAR
eLastState 	:= eState;
eState 		:= HALTED;

FOR idx := 0 TO 1 DO
	Components[idx].M_Halt();
END_FOR;
END_METHOD

{warning 'add method implementation '}
METHOD M_Reset : BOOL
END_METHOD

{warning 'add method implementation '}
METHOD M_Resume : BOOL

VAR
	idx: INT;
END_VAR
FOR idx := 0 TO 2 DO
	Components[idx].M_Resume();
END_FOR;

CASE eState OF
	HALTED:		eState := eLastState;
	DONE:		eState := READY;
END_CASE
END_METHOD

{warning 'add method implementation '}
METHOD M_Stop : BOOL
END_METHOD

END_FUNCTION_BLOCK

// ---- POUs/FB_Module_CoilPusher.TcPOU
FUNCTION_BLOCK FB_Module_CoilPusher IMPLEMENTS I_Module
VAR_INPUT
	bEnable		: BOOL;
END_VAR
VAR_OUTPUT
END_VAR
VAR
	Components	: ARRAY [0..1] OF I_Component;
	
	fbServo		: FB_Component_ServoMotor;
	fbSensor	: FB_Component_InductiveSensor;
	
	idx			: INT;
END_VAR

IF bEnable THEN
	fbServo(
		bEnable 			:= TRUE, 
		bHomingSensor 		:= GVL.bCoilTranslate, 
		bHomingSpeed 		:= 0, 
		uMaxRPM 			:= 3000,
		bSetCounterDone		:= GVL.bSetCounterDoneServo1,
		rGearRatio			:= 1,
		dCountServo			:= GVL.dCountServo1,
		bSetCounter			:= GVL.dSetCounterServo1,
		dSetCounterValue	:= GVL.dSetCounterValueServo1,
		bEnableDrive 		:= GVL.b603Enable, 
		uAnalogOut 			:= GVL.aOutServo1);
	
	fbSensor(
		bRawSignal			:= GVL.bCoilTranslate,
		tDebounce			:= T#5MS,
		tTimeout			:= T#5MS,
		sName				:= 'translate coil sens',
		bEnable				:= TRUE);
	
	Components[0]	:= fbServo;
	Components[1]	:= fbSensor;
	
	FOR idx := 0 TO 1 DO
    	Components[idx].M_Start();
	END_FOR;
END_IF

METHOD M_Extend : BOOL
VAR_INPUT
	uPos	: INT;
END_VAR
IF bEnable THEN
	M_Extend := fbServo.M_Goto(30000, 2, 500);
END_IF
END_METHOD

{warning 'add method implementation '}
METHOD M_Halt : BOOL
END_METHOD

METHOD M_Home : BOOL
VAR_INPUT
END_VAR
IF bEnable THEN
	IF fbSensor.bSensorActive THEN
		fbServo.M_SetSpeed(0);
		fbServo.M_DisableDrive();
		IF fbServo.M_SetCounter(0) THEN
			M_Home := TRUE;
		END_IF
	ELSE
		fbServo.M_EnableDrive();
		fbServo.M_SetSpeed(-2);
	END_IF
END_IF
END_METHOD

{warning 'add method implementation '}
METHOD M_Start : BOOL
END_METHOD

{warning 'add method implementation '}
METHOD M_Stop : BOOL
END_METHOD

END_FUNCTION_BLOCK

// ---- POUs/FB_Section_Cutter.TcPOU
FUNCTION_BLOCK FB_Section_Cutter IMPLEMENTS  I_Section
VAR_INPUT
	bEnable				: BOOL;
END_VAR
VAR_OUTPUT
END_VAR
VAR
	Components				: ARRAY [0..12] OF I_Component;	

	fbModule4posArm			: FB_Module_4posArm_Old;
	fbWireCutter			: FB_Component_SingleValve;
	
	fbWirePusher			: FB_Component_SingleValve;
	fbWirePusherExtended	: FB_Component_ReedSwitch;	//
	fbWirePusherRetracted	: FB_Component_ReedSwitch;	//
	
	fbShortTransverse		: FB_Component_DualValve;
	fbShortTransExtended	: FB_Component_ReedSwitch;	//
	fbShortTransRetracted	: FB_Component_ReedSwitch;	//
	
	fbLongTransverse		: FB_Component_DualValve;
	fbLongTransExtended		: FB_Component_ReedSwitch;	//
	fbLongTransRetracted	: FB_Component_ReedSwitch;	//
	
	fbWireClamp				: FB_Component_DualValve;
	fbWireClampRetracted	: FB_Component_ReedSwitch;	//
	
	fbWireClampActuator		: FB_Component_DualValve;
	idx: INT;
END_VAR

IF bEnable THEN
	fbModule4posArm(bEnable := TRUE);
	fbWireCutter(sName := 'wire cutter', bEnable := TRUE, bOutput := GVL.bCutWire);
	
	fbWirePusher(sName := 'wire cutter', bEnable := TRUE, bOutput := GVL.bWirePusherForward);
	fbWirePusherExtended(bRawSignal  := GVL.bWirePusherEngaged,		tDebounce := T#0MS, tTimeout := T#0MS, sName := 'wire pusher extended reed', bEnable := TRUE);
	fbWirePusherRetracted(bRawSignal := GVL.bWirePusherDisengaged, 	tDebounce := T#0MS, tTimeout := T#0MS, sName := 'wire pusher retracted reed',bEnable := TRUE);
		
	fbShortTransverse(sName := 'short transverse', bEnable := TRUE, bOutputA := GVL.bExtendWireHolderTransverse2, bOutputB := GVL.bRetractWireHolderTransverse2);
	fbShortTransExtended(bRawSignal  := GVL.bWireClampTransverse1Extended, tDebounce := T#0MS, tTimeout := T#0MS, sName := 'short trans extended reed', bEnable := TRUE);
	fbShortTransRetracted(bRawSignal := GVL.bWireClampTransverse1Retracted,tDebounce := T#0MS, tTimeout := T#0MS, sName := 'short trans retracted reed',bEnable := TRUE);	
	
	fbLongTransverse(sName := 'long transverse', bEnable := TRUE, bOutputA := GVL.bExtendWireHolderTransverse1, bOutputB := GVL.bRetractWireHolderTransverse1);
	fbLongTransExtended(bRawSignal  := GVL.bWireClampTransverse2Extended, tDebounce := T#0MS, tTimeout := T#0MS, sName := 'short trans extended reed', bEnable := TRUE);
	fbLongTransRetracted(bRawSignal := GVL.bWireClampTransverse2Retracted,tDebounce := T#0MS, tTimeout := T#0MS, sName := 'short trans retracted reed',bEnable := TRUE);
		
	fbWireClamp(sName := 'wire clamp', bEnable := TRUE, bOutputA := GVL.bEngageWireClamp, bOutputB := GVL.bReleaseWireClamp);
	fbWireClampRetracted(bRawSignal := GVL.bWireClampRetracted,tDebounce := T#0MS, tTimeout := T#0MS, sName := 'wire clamp retracted',bEnable := TRUE);
	
	fbWireClampActuator(sName := 'wire clamp actuator', bEnable := TRUE, bOutputA := GVL.bExtendWireClamp, bOutputB := GVL.bRetractWireClamp);
		
	Components[0]		:= fbWireCutter;
	Components[1]		:= fbWirePusher;
	Components[2]		:= fbWirePusherExtended;
	Components[3]		:= fbWirePusherRetracted;
	Components[4]		:= fbShortTransverse;
	Components[5]		:= fbShortTransExtended;
	Components[6]		:= fbShortTransRetracted;
	Components[7]		:= fbLongTransverse;
	Components[8]		:= fbLongTransExtended;
	Components[9]		:= fbLongTransRetracted;
	Components[10]		:= fbWireClamp;
	Components[11]		:= fbWireClampRetracted;
	Components[12]		:= fbWireClampActuator;
	
	fbModule4posArm.M_Start();
	FOR idx := 0 TO 12 DO
    	Components[idx].M_Start();
	END_FOR;
END_IF

METHOD M_GotoPos1 : BOOL
VAR_INPUT
END_VAR
IF bEnable THEN
	fbWirePusher.M_Retract();
	fbWireClamp.M_Extend();
	fbWireClampActuator.M_Extend();
	fbShortTransverse.M_Extend();
	fbLongTransverse.M_Retract();
	
	IF 	fbModule4posArm.M_Goto(2) 				 
		AND NOT fbWireClampRetracted.bSensorActive 
		AND fbShortTransExtended.bSensorActive
		AND fbLongTransRetracted.bSensorActive
		AND fbWirePusherRetracted.bSensorActive THEN
		
		fbWireClamp.M_Hold();
		fbWireClampActuator.M_Hold();
		fbShortTransverse.M_Hold();
		fbLongTransverse.M_Hold();
		M_GotoPos1 := TRUE;
	END_IF
END_IF
END_METHOD

{warning 'add method implementation '}
METHOD M_Halt : BOOL
END_METHOD

METHOD M_Seq_1 : BOOL
VAR_INPUT
END_VAR
IF fbLongTransExtended.bSensorActive THEN
	fbLongTransverse.M_Hold();
	
	IF fbWireClampRetracted.bSensorActive THEN
		fbWireClampActuator.M_Hold();		
		fbWireClamp.M_Hold();
		fbWirePusher.M_Extend();
		IF fbModule4posArm.M_Goto(1) THEN
			M_Seq_1 := TRUE;
		END_IF
	ELSE
		fbWireClampActuator.M_Retract();
		fbWireClamp.M_Retract();
	END_IF
ELSE
	fbLongTransverse.M_Extend();
END_IF
END_METHOD

METHOD M_Seq_2 : BOOL
VAR_INPUT
END_VAR
IF fbLongTransRetracted.bSensorActive THEN
	fbLongTransverse.M_Hold();
	fbWirePusher.M_Retract();
	M_Seq_2 := TRUE;
ELSE
	fbLongTransverse.M_Retract();
END_IF
END_METHOD

{warning 'add method implementation '}
METHOD M_Start : BOOL
END_METHOD

{warning 'add method implementation '}
METHOD M_Stop : BOOL
END_METHOD

END_FUNCTION_BLOCK

// ---- POUs/FB_Section_ToolStation_Old.TcPOU
FUNCTION_BLOCK FB_Section_ToolStation_Old IMPLEMENTS I_Section
VAR_INPUT
	bEnable					: BOOL;
END_VAR
VAR_OUTPUT
END_VAR
VAR
	bTriggerToolRotation	: BOOL;
	Modules					: ARRAY [0..2] OF I_Module;	

	fbCoilHolder			: FB_Module_CoilHolder_Old;
	fbToolHolderDoor		: FB_Module_ToolHolderDoor_Old;
	fbToolHolder			: FB_Module_ToolHolder_Old;
	
	idx						: INT;
END_VAR

IF bEnable THEN
	fbCoilHolder(bEnable 			:= TRUE);
	fbToolHolderDoor(bEnable 		:= TRUE);
	fbToolHolder(
			bEnable 				:= TRUE, 
			bToolRotationBtn 		:= bTriggerToolRotation, 
			bToolRotationBtnLight 	:= GVL.bToolingRotationBtnLight);
	
	Modules[0]	:= fbCoilHolder;
	Modules[1]	:= fbToolHolderDoor;
	Modules[2]	:= fbToolHolder;
	
	FOR idx := 0 TO 2 DO
    	Modules[idx].M_Start();
	END_FOR;
	
	IF GVL.bToolingRotationBtn AND fbToolHolderDoor.bDoorUp THEN
		bTriggerToolRotation := TRUE;
	ELSE
		bTriggerToolRotation := FALSE;
	END_IF
END_IF

METHOD M_CloseDoor : BOOL
VAR_INPUT
END_VAR
IF bEnable THEN
	M_CloseDoor := fbToolHolderDoor.M_Up();
END_IF
END_METHOD

METHOD M_Goto : BOOL
VAR_INPUT
	nTargetIndex: INT;
END_VAR

VAR
END_VAR
IF bEnable THEN
	M_Goto := fbCoilHolder.M_GoTo(nTargetIndex := nTargetIndex);
END_IF
END_METHOD

{warning 'add method implementation '}
METHOD M_Halt : BOOL
END_METHOD

METHOD M_OpenDoor : BOOL
VAR_INPUT
END_VAR
IF bEnable THEN
	M_OpenDoor := fbToolHolderDoor.M_Down();
END_IF
END_METHOD

{warning 'add method implementation '}
METHOD M_Start : BOOL
END_METHOD

{warning 'add method implementation '}
METHOD M_Stop : BOOL
END_METHOD

END_FUNCTION_BLOCK

// ---- POUs/MAIN.TcPOU
PROGRAM MAIN
VAR
	fbServo		: FB_Component_Servo;
	func		: INT;
	target		: INT := 1;
	set			: BOOL;
	hal			: BOOL;
	res			: BOOL;
	
	fbPiston	: FB_Module_ToolHolder;
	bEn: BOOL;
	
	tTimer		: TON;
END_VAR

// GVL.bUnlockCoilHolder

fbPiston(sName := '', tTimeout := T#5S);
tTimer(PT := T#1S);

IF bEn AND NOT fbPiston.bEnabled THEN
	fbPiston.M_Enable();
	bEn := FALSE;
END_IF 

IF set THEN
	CASE func OF
			//tTimer(IN := TRUE);
		2: fbPiston.M_Halt();
		3: fbPiston.M_Resume();
		4: fbPiston.M_Disable();
	END_CASE
	set := FALSE;
END_IF

IF tTimer.Q THEN
	tTimer(IN := FALSE);
	fbPiston.M_Halt();
END_IF


(*fbServo(
	sName 			:= '',
	tTimeout 		:= T#0MS,
	uMaxRPMservo 	:= 3000,
	rGearRatio 		:= 2.25,
	bRTO 			:= GVL.bReadyToOperate614,
	bEnableDrive 	:= GVL.b614Enable,
	bResetDrive 	:= GVL.bResetServosErrors,
	uAnalogOut 		:= GVL.aOutServo2);

IF NOT fbServo.bEnabled THEN
	fbServo.M_Enable();
END_IF

IF set THEN
	fbServo.M_SetAcceleration(uRPMperSec := 50);
	fbServo.M_SetRPMlimit(RPM := 700);
	fbServo.M_SetTargetRPM(target);
	set := FALSE;
END_IF

IF NOT GVL.bFeedBackSafetyRelay THEN
	IF NOT (fbServo.eState = E_State.HALTED) THEN
		fbServo.M_Halt();
		hal := FALSE;
	END_IF
	
END_IF

IF res THEN
	fbServo.M_Resume();
	res := FALSE;
END_IF*)

END_PROGRAM
